IF(PWM_Y39_SET<=300)THEN
	PWM_Y39_SET :=0;
END_IF
IF(PWM_Y40_SET<=300)THEN
	PWM_Y40_SET :=0;
END_IF

END_PROGRAM

// StandardPLC/Application/SaveEngine/SaveEngineMode_12
PROGRAM SaveEngineMode_12
VAR
	PAR_Y1_PosFull:UINT:=600;
END_VAR

(*******************节能控制阀主阀主泵输出执行**************************)
	
//ELSIF(GVL_SaveEngine.SaveEngineMode=12)THEN//节能下降回至中位模式,
	//GVL_SaveEngine.Y72OutPutState:=0;
	//GVL_SaveEngine.Y71OutPutState:=0;
	(****先关Y72再关Y71减少回中位时M1压力冲击****)
GVL_SaveEngine.Y72OutPutState:=0;
IF Mode12Timer>0 THEN
	GVL_SaveEngine.Y71OutPutState:=0;
END_IF
	Y73:=TRUE;
	
PWM_Y7_SET_Target:=0;
PWM_Y9_SET_Target:=0;
PWM_Y8_SET_Target:=0;
PWM_Y10_SET_Target:=0;
RAMP7(
	IN:=WORD_TO_INT(PWM_Y7_SET_Target), 
	ASCEND:= R_RAMP_mainwinch, 
	DESCEND:= F_RAMP_mainwinch_up, 
	TIMEBASE:=TIMEBASE_mainwinch , 
	RESET:=FALSE , 
	OUT=>(PWM_Y7_SET_Target1));
IF(PWM_Y7_SET_Target1>=400) THEN
	Curve_input:=TO_UINT(PWM_Y7_SET_Target1 - 400);
	IF(Curve_input>900) THEN
		Curve_input:=900;
	END_IF
	curve7(input:=REAL_TO_UINT(UINT_TO_REAL(Curve_input)*72.8),Zero:=FALSE,Full:=FALSE,
		   PAR_Progression:=Curve_Par,OutputEnable:=TRUE);
	PWM_Y7_SET:=PAR_Valve1_NegFull + REAL_TO_UINT(UINT_TO_REAL(curve7.Output)/72.8);
ELSE
	PWM_Y7_SET:=0;
END_IF
	
RAMP8(
	IN:=WORD_TO_INT(PWM_Y8_SET_Target), 
	ASCEND:= R_RAMP_mainwinch, 
	DESCEND:= F_RAMP_mainwinch_down, 
	TIMEBASE:=TIMEBASE_mainwinch , 
	RESET:=FALSE , 
	OUT=>(PWM_Y8_SET_Target1));
IF(PWM_Y8_SET_Target1>=400) THEN
	Curve_input:=TO_UINT(PWM_Y8_SET_Target1 - 400);
	IF(Curve_input>900) THEN
		Curve_input:=900;
	END_IF
	curve8(input:=REAL_TO_UINT(UINT_TO_REAL(Curve_input)*72.8),Zero:=FALSE,Full:=FALSE,
		   PAR_Progression:=Curve_Par,OutputEnable:=TRUE);
	PWM_Y8_SET:=PAR_Valve1_NegFull + REAL_TO_UINT(UINT_TO_REAL(curve8.Output)/72.8);
ELSE
	PWM_Y8_SET:=0;
END_IF
	RAMP9(
	IN:=WORD_TO_INT(PWM_Y9_SET_Target), 
	ASCEND:= R_RAMP_mainwinch, 
	DESCEND:= F_RAMP_mainwinch_up, 
	TIMEBASE:=TIMEBASE_mainwinch , 
	RESET:=FALSE , 
	OUT=>(PWM_Y9_SET_Target1));
IF(PWM_Y9_SET_Target1>=400) THEN
	Curve_input:=TO_UINT(PWM_Y9_SET_Target1 - 400);
	IF(Curve_input>900) THEN
		Curve_input:=900;
	END_IF
	curve9(input:=REAL_TO_UINT(UINT_TO_REAL(Curve_input)*72.8),Zero:=FALSE,Full:=FALSE,
		   PAR_Progression:=Curve_Par,OutputEnable:=TRUE);
	PWM_Y9_SET:=PAR_Valve1_NegFull + REAL_TO_UINT(UINT_TO_REAL(curve9.Output)/72.8);
ELSE
	PWM_Y9_SET:=0;
END_IF

RAMP10(
	IN:=WORD_TO_INT(PWM_Y10_SET_Target), 
	ASCEND:= R_RAMP_mainwinch, 
	DESCEND:= F_RAMP_mainwinch_down, 
	TIMEBASE:=TIMEBASE_mainwinch , 
	RESET:=FALSE , 
	OUT=>(PWM_Y10_SET_Target1));
IF(PWM_Y10_SET_Target1>=400) THEN
	Curve_input:=TO_UINT(PWM_Y10_SET_Target1 - 400);
	IF(Curve_input>900) THEN
		Curve_input:=900;
	END_IF
	curve10(input:=REAL_TO_UINT(UINT_TO_REAL(Curve_input)*72.8),Zero:=FALSE,Full:=FALSE,
		   PAR_Progression:=Curve_Par,OutputEnable:=TRUE);
	PWM_Y10_SET:=PAR_Valve1_NegFull + REAL_TO_UINT(UINT_TO_REAL(curve10.Output)/72.8);
ELSE
	PWM_Y10_SET:=0;
END_IF
//Y7 8 9 10范围限制
IF(PWM_Y7_SET>1300)THEN
	PWM_Y7_SET :=1300;
END_IF
IF(PWM_Y8_SET>1300)THEN
	PWM_Y8_SET :=1300;
END_IF
IF(PWM_Y9_SET>1300)THEN
	PWM_Y9_SET :=1300;
END_IF
IF(PWM_Y10_SET>1300)THEN
	PWM_Y10_SET :=1300;
END_IF

IF(PWM_Y7_SET<=300)THEN
	PWM_Y7_SET :=0;
END_IF
IF(PWM_Y8_SET<=300)THEN
	PWM_Y8_SET :=0;
END_IF
IF(PWM_Y9_SET<=300)THEN
	PWM_Y9_SET :=0;
END_IF
IF(PWM_Y10_SET<=300)THEN
	PWM_Y10_SET :=0;
END_IF
	
	
DOH_Y56:=FALSE;
PWM_Y33_SET_Target:=417;//110排量
PWM_Y33_SET := PWM_Y33_SET_Target;
//PWM_Y7_SET:=0;
//PWM_Y9_SET:=0;
//PWM_Y8_SET:=0;
//PWM_Y10_SET:=0;
PWM_Y1_SET:=0;//PWM_Y1_Target 直接给输出 去除中间变量
PWM_Y2_SET:=0; //PWM_Y2_Target 

PWM_Y39_SET_Target:=0;
PWM_Y40_SET_Target:=0;
RAMP19(
IN:=WORD_TO_INT(PWM_Y39_SET_Target), 
ASCEND:= R_RAMP_xiehe, 
DESCEND:= F_RAMP_xiehe, 
TIMEBASE:=TIMEBASE_xiehe , 
RESET:=FALSE , 
OUT=>(PWM_Y39_SET_Target1));
IF(PWM_Y39_SET_Target1>=400) THEN
Curve_input:=TO_UINT(PWM_Y39_SET_Target1 - 400);
IF(Curve_input>900) THEN
	Curve_input:=900;
END_IF
curve19(input:=REAL_TO_UINT(UINT_TO_REAL(Curve_input)*72.8),Zero:=FALSE,Full:=FALSE,
	   PAR_Progression:=Curve_Par1,OutputEnable:=TRUE);
PWM_Y39_SET:=PAR_Valve1_NegFull + REAL_TO_UINT(UINT_TO_REAL(curve19.Output)/72.8);
ELSE
PWM_Y39_SET:=0;
END_IF


RAMP20(
IN:=WORD_TO_INT(PWM_Y40_SET_Target), 
ASCEND:= R_RAMP_xiehe, 
DESCEND:= F_RAMP_xiehe, 
TIMEBASE:=TIMEBASE_xiehe , 
RESET:=FALSE , 
OUT=>(PWM_Y40_SET_Target1));
IF(PWM_Y40_SET_Target1>=400) THEN
Curve_input:=TO_UINT(PWM_Y40_SET_Target1 - 400);
IF(Curve_input>900) THEN
	Curve_input:=900;
END_IF
curve20(input:=REAL_TO_UINT(UINT_TO_REAL(Curve_input)*72.8),Zero:=FALSE,Full:=FALSE,
	   PAR_Progression:=Curve_Par1,OutputEnable:=TRUE);
PWM_Y40_SET:=PAR_Valve1_NegFull + REAL_TO_UINT(UINT_TO_REAL(curve20.Output)/72.8);
ELSE
PWM_Y40_SET:=0;
END_IF

IF(PWM_Y39_SET>1300)THEN
PWM_Y39_SET :=1300;
END_IF
IF(PWM_Y40_SET>1300)THEN
PWM_Y40_SET :=1300;
END_IF

IF(PWM_Y39_SET<=300)THEN
PWM_Y39_SET :=0;
END_IF
IF(PWM_Y40_SET<=300)THEN
PWM_Y40_SET :=0;
END_IF

(*
PWM_Y8_SET:=REAL_TO_UINT(INT_TO_REAL(PWM_JOYY_L_UP_1)/1000*(PAR_Valve1_PosFull-PAR_Valve1_NegFull)+PAR_Valve1_NegFull);
PWM_Y10_SET:=REAL_TO_UINT(INT_TO_REAL(PWM_JOYY_L_UP_1)/1000*(PAR_Valve2_PosFull-PAR_Valve2_NegFull)+PAR_Valve2_NegFull);
PWM_Y1_Target:=REAL_TO_UINT(INT_TO_REAL(PWM_JOYY_L_UP_1)/1000*(PAR_Y1_PosFull-PAR_Y1_NegFull)+PAR_Y1_NegFull);
PWM_Y2_Target:=REAL_TO_UINT(INT_TO_REAL(PWM_JOYY_L_UP_1)/1000*(PAR_Y1_PosFull-PAR_Y2_NegFull)+PAR_Y2_NegFull);
*)
(*  //Y33输出处理
IF PWM_Y33_SET>=PWM_Y33_SET_Target THEN
PWM_Y33_SET := PWM_Y33_SET_Target;
END_IF
	
IF(PWM_Y33_SET<PWM_Y33_SET_Target) THEN
	PWM_Y33_SET:=REAL_TO_UINT(UINT_TO_REAL(PWM_Y33_SET)+JianGE6);
END_IF

IF DIL_SQ3 THEN
	PWM_Y33_SET:=0;
END_IF
*)	
(*主泵功率控制*)

//区分发动机转速
MainPump_Pressure_Taget1450:=PAR_NegFull_x;
MainPump_Pressure_Taget1600:=PAR_PosFull_x;
MainPump_Pressure_Taget1750:=PAR_Zero_x;
IF EngineSpeedTarget<=1080 THEN SPEED_CASE:=1;
ELSIF EngineSpeedTarget>1080 AND EngineSpeedTarget<=1300 THEN SPEED_CASE:=2;
ELSIF EngineSpeedTarget>1300 AND EngineSpeedTarget<=1520 THEN SPEED_CASE:=3;
ELSIF EngineSpeedTarget>1520 AND EngineSpeedTarget<=1680 THEN SPEED_CASE:=4;
ELSIF EngineSpeedTarget>1680 AND EngineSpeedTarget<=1820 THEN SPEED_CASE:=5;
ELSIF EngineSpeedTarget>1820 THEN SPEED_CASE:=6;;END_IF
//不同转速下的发动机最大功率*)
CASE SPEED_CASE OF
1:  Enginer_Power:=135;
2:  Enginer_Power:=174;
3:  Enginer_Power:=200;
4:  Enginer_Power:=230;
5:  Enginer_Power:=250;
6:  Enginer_Power:=261;
END_CASE
//不同转速下的压力值
IF(CANO_Fubeng_Press>100)THEN
	CASE SPEED_CASE OF
	1:MainPump_Pressure_Taget:=MainPump_Pressure_Taget1000-HELIU_Press_Target1000;
	2:MainPump_Pressure_Taget:=MainPump_Pressure_Taget1200-HELIU_Press_Target1200;
	3:MainPump_Pressure_Taget:=MainPump_Pressure_Taget1450-HELIU_Press_Target1400;
	4:MainPump_Pressure_Taget:=MainPump_Pressure_Taget1600-HELIU_Press_Target1600;
	5:MainPump_Pressure_Taget:=MainPump_Pressure_Taget1750-HELIU_Press_Target1800;
	6:MainPump_Pressure_Taget:=MainPump_Pressure_Taget1900-HELIU_Press_Target1900;
	END_CASE
ELSE
	CASE SPEED_CASE OF
	1:MainPump_Pressure_Taget:=MainPump_Pressure_Taget1000;
	2:MainPump_Pressure_Taget:=MainPump_Pressure_Taget1200;
	3:MainPump_Pressure_Taget:=MainPump_Pressure_Taget1450;
	4:MainPump_Pressure_Taget:=MainPump_Pressure_Taget1600;
	5:MainPump_Pressure_Taget:=MainPump_Pressure_Taget1750;
	6:MainPump_Pressure_Taget:=MainPump_Pressure_Taget1900;
	END_CASE		
END_IF

IF( CANI_ECOSwitch) THEN
	CASE SPEED_CASE OF
	1:MainPump_Pressure_Taget:=MainPump_Pressure_Taget1000-ECO_Press_Target1000;
	2:MainPump_Pressure_Taget:=MainPump_Pressure_Taget1200-ECO_Press_Target1200;
	3:MainPump_Pressure_Taget:=MainPump_Pressure_Taget1450-ECO_Press_Target1400;
	4:MainPump_Pressure_Taget:=MainPump_Pressure_Taget1600-ECO_Press_Target1600;
	5:MainPump_Pressure_Taget:=MainPump_Pressure_Taget1750-ECO_Press_Target1800;
	6:MainPump_Pressure_Taget:=MainPump_Pressure_Taget1900-ECO_Press_Target1900;
	END_CASE
END_IF
MainPump_Pressure:=CANO_MainPUMP_Press1+CANO_MainPUMP_Press2;
//消除滤波
MainPump_Pressure_Subtract:= UINT_TO_INT(MainPump_Pressure-MainPump_Pressure_last1);


//大范围波动
IF MainPump_Pressure_Subtract>270 OR MainPump_Pressure_Subtract<-270 THEN
	Subtract:=TRUE;
ELSE
	Subtract:=FALSE;	
END_IF
	TIME_LvBo4(IN:=Subtract,PT:=T#10MS);
	
IF(TIME_LvBo4.Q)  AND (CANO_MainPUMP_Press1>210) THEN 
		MainPump_Pressure_ChangeBool1:=TRUE;
END_IF
	TIME_LvBo1(IN:=MainPump_Pressure_ChangeBool1,PT:=T#2S);
IF(TIME_LvBo1.Q) THEN
	MainPump_Pressure_ChangeBool1 :=FALSE;
END_IF

IF(MainPump_Pressure_ChangeBool1) AND (MainPump_Pressure>MainPump_Pressure_last1) THEN 
	MainPump_Pressure_last1:=MainPump_Pressure;
END_IF

//小范围波动
t_powertime:=TO_TIME(PAR_DeadBand_x);
IF (NOT MainPump_Pressure_ChangeBool1) THEN
	IF(MainPump_Pressure_Subtract>40 OR MainPump_Pressure_Subtract<-40)THEN 
		MainPump_Pressure_ChangeBool:=TRUE;
	ELSE
		MainPump_Pressure_ChangeBool:=FALSE;
	END_IF

	TIME_LvBo2(IN:=MainPump_Pressure_ChangeBool,PT:=t_powertime);
	IF(TIME_LvBo2.Q )THEN
		MainPump_Pressure_last1:=MainPump_Pressure;
	END_IF	
END_IF


IF PowerHead_move AND NOT(MainWinch_move) THEN
		JianGE2:=0.005;
ELSE
	IF(EngineSpeedTarget>1000 AND EngineSpeedTarget<1300)THEN
		JianGE2:=0.005;
	ELSE
		JianGE2:=0.005;
	END_IF
END_IF


IF MainPump_Pressure_last1>MainPump_Pressure_Taget THEN
	Pressure_Coe_Taget:=UINT_TO_REAL(MainPump_Pressure_Taget)/UINT_TO_REAL(MainPump_Pressure_last1);(*压力系数*)
ELSE
	Pressure_Coe_Taget:=1;
END_IF
Pressure_Coe := Pressure_Coe_Taget;


Pressure_Coe := 1;
IF MainPump_Pressure_last1>MainPump_Pressure_Taget  THEN
	IF(PWM_Y1_Target>=PAR_Y1_1_NegFull)THEN
		PWM_Y1_Target_OutPut:=REAL_TO_UINT(UINT_TO_REAL(PWM_Y1_Target-PAR_Y1_1_NegFull)*Pressure_Coe+PAR_Y1_1_NegFull);
	END_IF
	IF(PWM_Y2_Target>=PAR_Y1_1_NegFull)THEN
		PWM_Y2_Target_OutPut:=REAL_TO_UINT(UINT_TO_REAL(PWM_Y2_Target-PAR_Y1_1_NegFull)*Pressure_Coe+PAR_Y1_1_NegFull);
	END_IF
ELSE
	PWM_Y1_Target_OutPut:=PWM_Y1_Target;
	PWM_Y2_Target_OutPut:=PWM_Y2_Target;
END_IF

//PWM_Y1_Target_OutPut:=PWM_Y1_Target;
//PWM_Y2_Target_OutPut:=PWM_Y2_Target;
IF(EngineSpeedTarget>CANO_SPEED AND CANO_SPEED>400)THEN
	EngineSpeedSub:=EngineSpeedTarget - CANO_SPEED;
ELSE
	EngineSpeedSub:=0;
END_IF

IF(PWM_Y1_Target_OutPut<300)THEN PWM_Y1_Target_OutPut:=300;END_IF	
IF(PWM_Y2_Target_OutPut<300)THEN PWM_Y2_Target_OutPut:=300;END_IF

RAMP15_IN:=PWM_Y1_Target_OutPut;
RAMP16_IN:=PWM_Y2_Target_OutPut;
(*
IF MainWinch_move  OR  LeftMove_move OR RightMove_move THEN  
	TIMEBASE_pump:=T#1000MS;
	TIMEBASE_xiehe:=T#500MS;
ELSE
	TIMEBASE_pump:=T#400MS;
	TIMEBASE_xiehe:=T#200MS;
END_IF
t_PowerHead_move(IN:= MainWinch_move,PT:=T#2S);
IF t_PowerHead_move.Q THEN
	F_RAMP_pump:=x_t_PowerHead_move;
	R_RAMP_pump:=x2_t_PowerHead_move;
ELSE
	F_RAMP_pump:=1000;
	R_RAMP_pump:=300;
END_IF
*)
(*  12模式不需要斜坡
RAMP15(
	IN:=UINT_TO_INT(RAMP15_IN), 
	ASCEND:= 300, 
	DESCEND:= 300, 
	TIMEBASE:=T#1000MS , 
	RESET:=FALSE , 
	OUT=>(PWM_Y1_SET));
	
RAMP16(
	IN:=UINT_TO_INT(RAMP16_IN), 
	ASCEND:= 300, 
	DESCEND:= 300, 
	TIMEBASE:=T#1000MS , 
	RESET:=FALSE , 
	OUT=>(PWM_Y2_SET));

*)

	CASE SPEED_CASE OF
                1:F_RAMP_pump:=1500; R_RAMP_pump:=100;                  
                2: 		IF MainWinch_move AND (JiaYa_move OR CANO_JiayaPressure>80)  THEN    //3泵同时起压时，降低主泵的加载速度，避免掉速熄火
                                F_RAMP_pump:=1500; R_RAMP_pump:=100;
                        ELSE
                                F_RAMP_pump:=1500; R_RAMP_pump:=100;//从200降
                                IF  PWM_JOYY_L_UP>10 THEN
                                 F_RAMP_pump:=1500; R_RAMP_pump:=200;
                                END_IF
                        END_IF            
                3:
                        IF MainWinch_move AND (JiaYa_move OR CANO_JiayaPressure>80)  THEN    //3泵同时起压时，降低主泵的加载速度，避免掉速熄火
                                F_RAMP_pump:=1500; R_RAMP_pump:=150;
                        ELSE
                                F_RAMP_pump:=1500; R_RAMP_pump:=TO_INT(PAR_NegFull_y);
                                IF  PWM_JOYY_L_UP>10 THEN
                                 F_RAMP_pump:=1500; R_RAMP_pump:=300;
                                END_IF
                        END_IF                
                4:
                        IF MainWinch_move AND (JiaYa_move OR CANO_JiayaPressure>80)  THEN
                                F_RAMP_pump:=1500; R_RAMP_pump:=150;
                        ELSE
                                F_RAMP_pump:=1500; R_RAMP_pump:=TO_INT(PAR_PosFull_y);//从200降
                                IF  PWM_JOYY_L_UP>10 THEN
                                 F_RAMP_pump:=1500; R_RAMP_pump:=300;
                                END_IF
                        END_IF                                
                5:
                        IF MainWinch_move AND (JiaYa_move OR CANO_JiayaPressure>80)  THEN
                                F_RAMP_pump:=1500; R_RAMP_pump:=200;
                        ELSE
                                F_RAMP_pump:=1500; R_RAMP_pump:=TO_INT(PAR_Zero_y);
                                IF  PWM_JOYY_L_UP>10 THEN
                                 F_RAMP_pump:=1500; R_RAMP_pump:=300;
                                END_IF
                        END_IF                        
                6:		IF MainWinch_move AND (JiaYa_move OR CANO_JiayaPressure>80)  THEN
                                F_RAMP_pump:=1500; R_RAMP_pump:=200;
                        ELSE
                                F_RAMP_pump:=1500; R_RAMP_pump:=200;
                                IF  PWM_JOYY_L_UP>10 THEN
                                 F_RAMP_pump:=1500; R_RAMP_pump:=300;
                                END_IF
                        END_IF	
	END_CASE
(******斜坡增步长300 斜坡降步长300->400*****)	
RAMP15(
	IN:=UINT_TO_INT(RAMP15_IN), 
	ASCEND:= R_RAMP_pump, 
	DESCEND:= 1500, 
	TIMEBASE:=T#1000MS , 
	RESET:=FALSE , 
	OUT=>(PWM_Y1_SET));
(******减斜坡300->400*****)	
RAMP16(
	IN:=UINT_TO_INT(RAMP16_IN), 
	ASCEND:= R_RAMP_pump, 
	DESCEND:= 1500, 
	TIMEBASE:=T#1000MS , 
	RESET:=FALSE , 
	OUT=>(PWM_Y2_SET));

IF (NOT Rotation_move) AND (NOT MainWinch_move) AND (NOT PowerHead_move)
		AND (NOT JiaYa_move) AND (NOT ViceWinch_move)
		AND (NOT LeftMove_move) AND (NOT RightMove_move)  THEN
	PWM_Y1_Target:=0;
	PWM_Y2_Target:=0;
END_IF

IF PWM_Y1_SET<TO_INT(PAR_Y1_1_NegFull )THEN
	PWM_Y1_SET:=TO_INT(PAR_Y1_1_NegFull);
END_IF

IF PWM_Y2_SET<TO_INT(PAR_Y1_1_NegFull )THEN
	PWM_Y2_SET:=TO_INT(PAR_Y1_1_NegFull);
END_IF

IF(PWM_Y1_SET>1000) THEN
	PWM_Y1_SET := 300;
END_IF

IF(PWM_Y2_SET>1000) THEN
	PWM_Y2_SET := 300;
END_IF

END_PROGRAM

// StandardPLC/Application/SaveEngine/SaveEngineMode_9
PROGRAM SaveEngineMode_9
VAR
DI_PWM_JOYX_L: BOOL;
	DI_PWM_JOYY_L: BOOL;
	DI_PWM_JOYX_R: BOOL;
	DI_PWM_JOYY_R: BOOL;
	DI_PWM_JOY_Jiao_R: BOOL;
	DI_PWM_JOY_Jiao_L: BOOL;
	Rotation_move: BOOL;
	MainWinch_move:BOOL;
	PowerHead_move:BOOL;
	JiaYa_move: BOOL;
	LvZhang_move: BOOL;
	BianFu_move:BOOL;
	ViceWinch_move: BOOL;
	LeftMove_move:BOOL;
	RightMove_move:BOOL;
	SPEED_CASE:USINT;
	Enginer_Power:UINT;
	
	PWM_Y1_Target: UINT;	
	PWM_Y2_Target: UINT;	
	
	PWM_Y1_Target_MAX: UINT;
	PWM_Y2_Target_MAX: UINT;
	Hydraulic_Power2:UINT;
	Hydraulic_Power1:UINT;
	Hydraulic_Power:UINT;
	Enginer_Rat: UINT;
	MainPump_Pressure_Taget:UINT;
	Coe_valve: REAL;	
	MainPump_Pressure: UINT;
	Pressure_Coe: REAL;
	PWM_Y1_Target_1: UINT;
	Single_move:BOOL;
	PWM_Y1_Target_OutPut: UINT;
	PWM_Y2_Target_OutPut: UINT;
	PWM_Y34_SET_Target: UINT:=0;
	PWM_Y33_SET_Target: UINT:=1100;
	

	DonglitouBlink:BLINK;
	DonglitouBlink_biaozhi:BOOL;
	DOH_Y50_1: BOOL;
	Rotation_late:TOF;
	MainPump_Pressure_Taget1000:UINT:=220;
	MainPump_Pressure_Taget1200:UINT:=360;
	MainPump_Pressure_Taget1450:UINT:=420;
	MainPump_Pressure_Taget1600:UINT:=420;
	MainPump_Pressure_Taget1750:UINT:=400;
	MainPump_Pressure_Taget1900:UINT:=360;
	Pressure_Coe_Taget: REAL;
	JianGE1: REAL:=1;
	JianGE2: REAL:=0.005;
	JianGE3: REAL:=3;
	TIME_100ms:TON;
	MainPump_Pressure_last: UINT;
	MainPump_Pressure_last1: UINT;
	TIME_LvBo1:TON;
	TIME_LvBo2:TON;
	TIME_LvBo3:TON;
	MainPump_Pressure_Subtract: INT;
	MainPump_Pressure_ChangeBool: BOOL;
	MainPump_Pressure_ChangeBool1:BOOL;
	PWM_Y2_Target_fuhe: UINT;
	PWM_Y1_Target_fuhe: UINT;
	EngineSpeedSub: UINT;
	PWM_Y23_SET_Taget: UINT;
	PWM_Y24_SET_Taget: UINT;
	CANO_DonglitouPressure_last: UINT;
	DonglitouPressureSub:INT;
	DonglitouPressure_ChangeBool: BOOL;
	JieSuoBool: BOOL;
	ECO_Press_Target1000: UINT:=50;
	ECO_Press_Target1200: UINT:=50;
	ECO_Press_Target1400: UINT:=50;
	ECO_Press_Target1600: UINT:=50;
	ECO_Press_Target1800: UINT:=50;
	ECO_Press_Target1900: UINT:=50;
	
	HELIU_Press_Target1000: UINT:=80;
	HELIU_Press_Target1200: UINT:=80;
	HELIU_Press_Target1400: UINT:=80;
	HELIU_Press_Target1600: UINT:=80;
	HELIU_Press_Target1800: UINT:=80;
	HELIU_Press_Target1900: UINT:=80;
	PWM_Y2_Target_P: UINT;
	PWM_JOY_P_W: UINT;
	XISHU1: REAL:=0.6;
	BiaoZHI_MainWinchUp: BOOL;
	JianGE6:REAL:=2;
	PWM_Y5_SET_Target: UINT;
	PWM_Y6_SET_Target: UINT;
	PWM_Y15_SET_Target: UINT;
	PWM_Y16_SET_Target: UINT;
	PWM_Y5_SET_Target1: INT;
	PWM_Y6_SET_Target1: INT;
	PWM_Y15_SET_Target1: INT;
	PWM_Y16_SET_Target1: INT;
	PWM_Y8_SET_Target: UINT;
	PWM_Y10_SET_Target: UINT;
	PWM_Y7_SET_Target: UINT;
	PWM_Y9_SET_Target: UINT;
	PWM_Y8_SET_Target1: INT;
	PWM_Y10_SET_Target1: INT;
	PWM_Y7_SET_Target1: INT;
	PWM_Y9_SET_Target1: INT;
	JianGE7: UINT:=20;
	JianGE8: UINT:=3;
	PWM_Y39_SET_Target: UINT;
	PWM_Y40_SET_Target: UINT;
	ABS_JOY_1: INT;
	PWM_Y61_SET_Tatget: UINT;
	PWM_Y12_SET_Tatget: UINT;
	PWM_Y14_SET_Tatget: UINT;
	PWM_Y60_SET_Tatget: UINT;
	PWM_Y11_SET_Tatget: UINT;
	PWM_Y13_SET_Tatget: UINT;
	PWM_Y61_SET_Tatget1: INT;
	PWM_Y12_SET_Tatget1: INT;
	PWM_Y14_SET_Tatget1: INT;
	PWM_Y60_SET_Tatget1: INT;
	PWM_Y11_SET_Tatget1: INT;
	PWM_Y13_SET_Tatget1: INT;
	JianGE10: UINT:=25;
	yyyy: UINT;
	TIME_200ms:TON;
	TIME_400ms:TON;
	CANI_JOYX_R_last:UINT;
	Sub_Joyx_r: INT;
	Joyx_change_bool: BOOL;
	JianGE12: UINT:=30;
	Sub_Joyx_r_1: INT;
	BIAOzhi1: BOOL;
	R_TRIG_1:R_TRIG;
	R_TRIG_BOOL: BOOL;
	JianGE22: REAL;
	
	
	curve:curve_quxian;
	curve1:curve_quxian;
	curve2:curve_quxian;
	curve3:curve_quxian;
	curve4:curve_quxian;
	curve5:curve_quxian;
	curve6:curve_quxian;
	curve7:curve_quxian;
	curve8:curve_quxian;
	curve9:curve_quxian;
	curve10:curve_quxian;
	curve11:curve_quxian;
	curve12:curve_quxian;
	curve13:curve_quxian;
	curve14:curve_quxian;
	curve19:curve_quxian;
	curve20:curve_quxian;
	COUNTER : INT;
	JianGE13: UINT:=40;
	JianGE14: UINT:=40;
	RAMP:RAMP_INT;
	RAMP1:RAMP_INT;
	RAMP2:RAMP_INT;
	RAMP3:RAMP_INT;
	R_RAMP:INT:=400;
	F_RAMP:INT:=250;
	TIMEBASE:TIME:=T#200MS;
	PWM_Y7_SET_Target111: INT;
	YYYYYYY:BOOL;
	JIANGE1111: INT:=20;
	
	RAMP4:RAMP_INT;
	RAMP5:RAMP_INT;
	RAMP6:RAMP_INT;
	RAMP7:RAMP_INT;
	RAMP8:RAMP_INT;
	RAMP9:RAMP_INT;
	RAMP10:RAMP_INT;
	RAMP11:RAMP_INT;
	RAMP12:RAMP_INT;
	RAMP13:RAMP_INT;
	RAMP14:RAMP_INT;
	RAMP15:RAMP_INT;
	RAMP16:RAMP_INT;
	RAMP17:RAMP_INT;
	RAMP18:RAMP_INT;
	RAMP19:RAMP_INT;
	RAMP20:RAMP_INT;
	RAMP21:RAMP_INT;
	RAMP22:RAMP_INT;
	RAMP23:RAMP_INT;
	RAMP24:RAMP_INT;
	PWM_Y23_SET_Taget1:INT;
	PWM_Y24_SET_Taget1:INT;
	PWM_Y18_SET_Taget1:INT;
	PWM_Y18_SET_Taget:UINT;
	ASCEND_value2:INT;
	//2023 01 13 增加
	//行走动作斜坡值
	R_RAMP_traval:INT:=800;
	F_RAMP_traval:INT:=400;
	TIMEBASE_traval:TIME:=T#200MS;
	//动力头动作斜坡值
	R_RAMP_ratate:INT:=800;
	F_RAMP_ratate:INT:=800;
	TIMEBASE_ratate:TIME:=T#100MS;
	//主卷扬动作斜坡值
	R_RAMP_mainwinch:INT:=800;
	F_RAMP_mainwinch_up:INT:=400;
	F_RAMP_mainwinch_down:INT:=400;
	TIMEBASE_mainwinch:TIME:=T#200MS;
	//主泵排量斜坡值
	R_RAMP_pump:INT:=300;
	F_RAMP_pump:INT:=1000;
	TIMEBASE_pump:TIME:=T#1000MS;
	//卸荷阀斜坡值
	R_RAMP_xiehe:INT:=500;
	F_RAMP_xiehe:INT:=400;
	TIMEBASE_xiehe:TIME:=T#500MS;
	
	//直线阀斜坡值
	R_RAMP_zhixian:INT:=800;
	F_RAMP_zhixian:INT:=800;
	TIMEBASE_zhixian:TIME:=T#300MS;
		
	Subtract: BOOL;
	TIME_LvBo4:TON;
	Curve_input:UINT;
	Curve_Par: SINT:=0;
	Curve_Par1: SINT:=0;
	Move_JOY_FUHE: UINT;
	PWM_JOY_Jiao_L_UP1:UINT;
	PWM_JOY_Jiao_L_DOWN1:UINT;
	PWM_JOY_Jiao_R_UP1:UINT;
	PWM_JOY_Jiao_R_DOWN1:UINT;
	
	PWM_JOYX_R_UP_a:UINT;
	PWM_JOYX_R_UP_b:UINT;
	
	PWM_JOYX_R_DOWN_a:UINT;
	PWM_JOYX_R_DOWN_b:UINT;
	
	PWM_JOYY_L_DOWN_a:UINT;
	PWM_JOYY_L_DOWN_b:UINT;
	
	PWM_JOYY_L_UP_a:UINT;
	PWM_JOYY_L_UP_b:UINT;
	aaaa:UINT:=500;
	
	JOY_PAOTU:BOOL;
	
	JOY_PAOTU_tiaojian:BOOL;
	TIME_1000_1ms:ton;
	tempbool:BOOL;
	CANI_JOYX_R_last2:UINT;
	Sub_Joyx_r2:INT;
	JianGE11:REAL:=2;
	JianGE21:uint:=10;
	END_IFc: INT;
	x1:UINT:=8;
	x2:UINT:=8;
	PWM_JOY_JIAO:UINT;
	PWM_Y39_SET1:UINT;
	PWM_Y40_SET1:UINT;
	aaa: INT;
	TIME_50ms:TON;
	TIME_55ms:TOF;
	TIME_2000ms:TOF;
	start_move: BOOL;
	T1:TIME;
	TEMP1:UINT;
	X3: INT;
	X4: INT;
	liandong:BOOL;
	PWM_Y9_SET1:INT;
	PWM_Y10_SET1:INT;
	PWM_Y13_SET1:INT;
	PWM_Y14_SET1:INT;
	yanchi1:BOOL;
	yanchi_ton1:ton;
	RAMP15_IN:UINT;
	RAMP16_IN:UINT;
	Rtrig_d1:R_TRIG;
	Rtrig_d2:R_TRIG;
	
	Rtrig_DongLiTou1:R_TRIG;
	Rtrig_DongLiTou2:R_TRIG;
	Count_TIMES_Fanzhuan: UINT;
	Count_TIMES_Zhengzhuan: UINT;
	TIME_1000ms:TON;
	TIME_1000ms_TP:TON;
	Count_TIMES_Fanzhuan_LAST: UINT;
	Count_TIMES_Zhengzhuan_LAST: UINT;
	Paotu_Modle: BOOL;
	PaoTU_biaozhi: BOOL;
	TIMEBASE_D: TIME;
	PWM_Y39_SET_Target1:INT;
	PWM_Y40_SET_Target1:INT;
	PWM_Y37_SET_Target:UINT;
	PWM_Y17_SET2:UINT;
	t_PowerHead_move:TON;
	x_t_PowerHead_move:INT:=10;//100-10
	x2_t_PowerHead_move:INT:=10;//100-10
	P_value:REAL;//动力头反转+主卷上提时的分流系数
	PWM_JOY_P:UINT;
	PWM_JOY_P1:UINT;
	PWM_JOY_P2:UINT;
	PWM_JOY_P3:UINT;
	PWM_JOY_P4:UINT;
	ASCEND_value:INT;
	ftp1:INT:=500;
	ftp2:INT:=100;
	t_powertime:TIME;
	
	P25_Flag:BOOL;
	P27_Flag:BOOL;
	P29_Flag:BOOL;
	P31_Flag:BOOL;
	PressLvBo_TON:TON;
	PressLvBo_TON1: TON;
	PressLvBo_TON2: TON;
	PressLvBo_TON3: TON;
	test: BYTE;
	testpaotu: UINT := 450;
END_VAR

//动力头反转与主卷上提时的分流系数值
(*IF CANO_ZhuJuanPressure<=100 THEN
	P_value:=TO_REAL(PAR_KI+40)/100.0;
ELSIF CANO_ZhuJuanPressure>100 AND  CANO_ZhuJuanPressure<=200 THEN
	P_value:=TO_REAL(PAR_KI+20)/100.0;
ELSE
	P_value:=TO_REAL(PAR_KI)/100;
END_IF*)
GVL_SaveEngine.Y72OutPutState:=0;
GVL_SaveEngine.Y71OutPutState:=0;
GVL_SaveEngine.Y73:=0;
P_value:=TO_REAL(PAR_KI)/100;  //出厂值设定为35
//喇叭
IF DI_LHandle_SB5 THEN
	DOH_Y59:=TRUE;
ELSE
	DOH_Y59:=FALSE;
END_IF
//延时断电
TIME_2000ms(IN:=DIH_power3,PT:=T#2S);
IF(TIME_2000ms.Q)THEN
	DOH_YS3:=TRUE;
ELSE
	DOH_YS3:=FALSE;
END_IF

//主卷上限位及解锁
IF(DI_LHandle_SB1 AND (NOT CANI_WorkModeSwitch))THEN
	JieSuoBool:=TRUE;
ELSE
	JieSuoBool:=FALSE;	
END_IF

IF DIL_SQ4 THEN
	IF(NOT JieSuoBool) THEN
		PWM_JOYY_L_DOWN:=0;
	END_IF
END_IF

//主卷下限位及解锁
//主卷下放限制
IF( CANO_MainWinchTension*100<PAR_MainWinchLaLi_Low) AND (NOT DI_LHandle_SB1) AND (CANI_WorkModeSwitch)THEN
	PWM_JOYY_L_UP:=0;
END_IF

TIME_50ms(in:=start_move,pt:=T1);
TIME_55ms(in:=start_move,pt:=T#500MS);
IF( LeftMove_move OR  RightMove_move  OR   MainWinch_move OR PowerHead_move OR ViceWinch_move )THEN
	start_move:=TRUE;
ELSE
	start_move:=FALSE;
END_IF
	 


IF NOT DIL_SQ3 THEN(*先导控制输入*)
	IF PWM_JOYX_L_UP>10 OR PWM_JOYX_L_DOWN>10 THEN  DI_PWM_JOYX_L := TRUE;ELSE DI_PWM_JOYX_L:=FALSE;END_IF(*左手柄左右动作*)
	IF PWM_JOYY_L_UP>10 OR PWM_JOYY_L_DOWN>10 THEN  DI_PWM_JOYY_L := TRUE;ELSE DI_PWM_JOYY_L:=FALSE;END_IF(*左手柄前后动作*)
	IF PWM_JOYX_R_UP>10 OR PWM_JOYX_R_DOWN>10 THEN  DI_PWM_JOYX_R := TRUE;ELSE DI_PWM_JOYX_R:=FALSE;END_IF(*右手柄左右动作*)
	IF PWM_JOYY_R_UP>10 OR PWM_JOYY_R_DOWN>10 THEN  DI_PWM_JOYY_R := TRUE;ELSE DI_PWM_JOYY_R:=FALSE;END_IF(*右手柄前后动作*)
	IF PWM_JOY_Jiao_L_UP>10 OR PWM_JOY_Jiao_L_DOWN>10 THEN  DI_PWM_JOY_Jiao_L:= TRUE;ELSE DI_PWM_JOY_Jiao_L:=FALSE;END_IF(*左脚踏前后动作*)
	IF PWM_JOY_Jiao_R_UP>10 OR PWM_JOY_Jiao_R_DOWN>10 THEN  DI_PWM_JOY_Jiao_R := TRUE;ELSE DI_PWM_JOY_Jiao_R:=FALSE;END_IF(*左脚踏左右动作*)
ELSE
	DI_PWM_JOYX_L:=FALSE;
	DI_PWM_JOYY_L:=FALSE;
	DI_PWM_JOYX_R:=FALSE;
	DI_PWM_JOYY_R:=FALSE;
	DI_PWM_JOY_Jiao_L:=FALSE;
	DI_PWM_JOY_Jiao_R:=FALSE;
END_IF

(*动作标志*)
IF DI_PWM_JOYY_L THEN MainWinch_move:=TRUE; ELSE MainWinch_move:=FALSE;END_IF(*主卷扬动作*)
IF DI_PWM_JOYX_L THEN Rotation_move:=TRUE; ELSE Rotation_move:=FALSE;END_IF(*回转动作*)
IF CANI_WorkModeSwitch THEN   (*作业挡情况下*)
	IF DI_PWM_JOYX_R THEN PowerHead_move:=TRUE;ELSE PowerHead_move:=FALSE;END_IF(*动力头回转动作*)
	IF DI_PWM_JOYY_R THEN JiaYa_move:=TRUE;ELSE JiaYa_move:=FALSE;END_IF(*动力头加压动作*)
	LvZhang_move:=FALSE;
	BianFu_move:=FALSE;
	ViceWinch_move:=FALSE;
	LeftMove_move:=FALSE;
	RightMove_move:=FALSE;
ELSE   (*调整档状态*)
	IF DI_PWM_JOYX_R THEN  LvZhang_move:=TRUE;ELSE LvZhang_move:=FALSE;END_IF(*L履带、张紧、支腿动作,M4阀*)
	(*LeftMove_move:=DI_PWM_JOY_Jiao_L;(*左行走动作*)
	RightMove_move:=DI_PWM_JOY_Jiao_R;*)(*右行走动作*)
	IF( PWM_JOY_Jiao_L_UP1>10 OR PWM_JOY_Jiao_L_DOWN1>10)  AND  DI_PWM_JOY_Jiao_L THEN
		LeftMove_move:=TRUE;
	ELSE
		LeftMove_move:=FALSE;
	END_IF
	IF( PWM_JOY_Jiao_R_UP1>10 OR PWM_JOY_Jiao_R_DOWN1>10)  AND  DI_PWM_JOY_Jiao_R THEN
		RightMove_move:=TRUE;
	ELSE
		RightMove_move:=FALSE;
	END_IF

	IF  DI_RHandle_SB5 THEN
		ViceWinch_move:=FALSE;
		IF  DI_PWM_JOYY_R  THEN BianFu_move:=TRUE;ELSE BianFu_move:=FALSE;END_IF(*变幅动作M4阀*)
	ELSE
		BianFu_move:=FALSE;
		IF DI_PWM_JOYY_R  THEN ViceWinch_move:=TRUE;ELSE ViceWinch_move:=FALSE;END_IF(*副卷扬动作M4阀*)
	END_IF
	PowerHead_move:=FALSE;
	JiaYa_move:=FALSE;
END_IF


(****主阀单动作标志****)
	IF (NOT MainWinch_move) AND (NOT PowerHead_move) AND (ViceWinch_move) THEN
		Single_move:=TRUE;
	ELSE
		Single_move:=FALSE;
	END_IF
	
//先导控制
IF(NOT DIL_SQ3) AND NOT VarGpsSystemLockedState THEN
	DOH_Y51:=TRUE;
ELSE
	DOH_Y51:=FALSE;
END_IF

//行走动作
(*脚踏阀偏差*)
IF   ((PWM_JOY_Jiao_L_UP-PWM_JOY_Jiao_R_UP)<200 OR(PWM_JOY_Jiao_R_UP-PWM_JOY_Jiao_L_UP)<200) THEN
	PWM_JOY_Jiao_L_UP1:=MAX(PWM_JOY_Jiao_L_UP,PWM_JOY_Jiao_R_UP);
	PWM_JOY_Jiao_R_UP1:=MAX(PWM_JOY_Jiao_L_UP,PWM_JOY_Jiao_R_UP);
ELSE
	PWM_JOY_Jiao_L_UP1:=PWM_JOY_Jiao_L_UP;
	PWM_JOY_Jiao_R_UP1:=PWM_JOY_Jiao_R_UP;
END_IF
IF   ((PWM_JOY_Jiao_L_DOWN-PWM_JOY_Jiao_R_DOWN)<200  OR  (PWM_JOY_Jiao_R_DOWN-PWM_JOY_Jiao_L_DOWN)<200 ) THEN
	PWM_JOY_Jiao_L_DOWN1:=MAX(PWM_JOY_Jiao_L_DOWN,PWM_JOY_Jiao_R_DOWN);
	PWM_JOY_Jiao_R_DOWN1:=MAX(PWM_JOY_Jiao_L_DOWN,PWM_JOY_Jiao_R_DOWN);
ELSE
	PWM_JOY_Jiao_L_DOWN1:=PWM_JOY_Jiao_L_DOWN;
	PWM_JOY_Jiao_R_DOWN1:=PWM_JOY_Jiao_R_DOWN;
END_IF

PWM_JOY_JIAO:=MAX(PWM_JOY_Jiao_L_UP1,PWM_JOY_Jiao_R_UP1,PWM_JOY_Jiao_L_DOWN1,PWM_JOY_Jiao_R_DOWN1);
liandong:=FALSE;
(*左行走*)
(*泵1   Y1   Y39控制右行走   Y15  16 *)
(*泵2   Y2 Y40 控制左行走    Y5  Y6*)
IF LeftMove_move THEN
	IF PWM_JOY_Jiao_L_UP1>10 THEN
		PWM_Y2_Target:=REAL_TO_UINT(UINT_TO_REAL(PWM_JOY_Jiao_L_UP1)/1000*(PAR_Y1_1_PosFull-PAR_Y1_1_NegFull)+PAR_Y1_1_NegFull);
		PWM_Y5_SET_Target:=REAL_TO_UINT(UINT_TO_REAL(PWM_JOY_Jiao_L_UP1)/1000*(PAR_Valve2_PosFull-PAR_Valve2_NegFull)+PAR_Valve2_NegFull);
		PWM_Y6_SET_Target:=0;	
	ELSIF PWM_JOY_Jiao_L_DOWN1>10 THEN
		PWM_Y2_Target:=REAL_TO_UINT(UINT_TO_REAL(PWM_JOY_Jiao_L_DOWN1)/1000*(PAR_Y1_1_PosFull-PAR_Y1_1_NegFull)+PAR_Y1_1_NegFull);
		PWM_Y6_SET_Target:=REAL_TO_UINT(UINT_TO_REAL(PWM_JOY_Jiao_L_DOWN1)/1000*(PAR_Valve2_PosFull-PAR_Valve2_NegFull)+PAR_Valve2_NegFull);
		PWM_Y5_SET_Target:=0;		
	END_IF
ELSE
	PWM_Y5_SET_Target:=0;
	PWM_Y6_SET_Target:=0;
END_IF
(*右行走*)
IF RightMove_move  THEN
	IF PWM_JOY_Jiao_R_UP1>10 THEN
		PWM_Y1_Target:=REAL_TO_UINT(UINT_TO_REAL(PWM_JOY_Jiao_R_UP1)/1000*(PAR_Y1_1_PosFull-PAR_Y1_1_NegFull)+PAR_Y1_1_NegFull);
		PWM_Y15_SET_Target:=REAL_TO_UINT(UINT_TO_REAL(PWM_JOY_Jiao_R_UP1)/1000*(PAR_Valve1_PosFull-PAR_Valve1_NegFull)+PAR_Valve1_NegFull);
		PWM_Y16_SET_Target:=0;
	
	ELSIF PWM_JOY_Jiao_R_DOWN1>10 THEN
		PWM_Y1_Target:=REAL_TO_UINT(UINT_TO_REAL(PWM_JOY_Jiao_R_DOWN1)/1000*(PAR_Y1_1_PosFull-PAR_Y1_1_NegFull)+PAR_Y1_1_NegFull);
		PWM_Y16_SET_Target:=REAL_TO_UINT(UINT_TO_REAL(PWM_JOY_Jiao_R_DOWN1)/1000*(PAR_Valve1_PosFull-PAR_Valve1_NegFull)+PAR_Valve1_NegFull);
		PWM_Y15_SET_Target:=0;
		
	END_IF
ELSE
	PWM_Y15_SET_Target:=0;
	PWM_Y16_SET_Target:=0;
END_IF

	//如有必要，可根据行走阀开关大小调整斜坡值
(*	IF(PWM_Y5_SET<1000  AND  PWM_Y5_SET>=900)THEN
			R_RAMP_traval:=100;
	ELSIF(PWM_Y5_SET<900 AND PWM_Y5_SET>=780)THEN
			R_RAMP_traval:=10;
	ELSE
			R_RAMP_traval:=250;
	END_IF
		
	IF(PWM_Y6_SET<1000  AND  PWM_Y6_SET>=900)THEN
			F_RAMP_traval:=100;		
	ELSIF(PWM_Y6_SET<900 AND PWM_Y6_SET>750 )THEN
			F_RAMP_traval:=15;
	ELSE
			F_RAMP_traval:=250;
	END_IF*)
	
(*行走动作缓冲*)
RAMP11(
	IN:=WORD_TO_INT(PWM_Y5_SET_Target), 
	ASCEND:= R_RAMP_traval, 
	DESCEND:= F_RAMP_traval, 
	TIMEBASE:=TIMEBASE_traval , 
	RESET:=FALSE , 
	OUT=>(PWM_Y5_SET_Target1));
IF(PWM_Y5_SET_Target1>=400) THEN
	Curve_input:=TO_UINT(PWM_Y5_SET_Target1 - 400);
	IF(Curve_input>900) THEN
		Curve_input:=900;
	END_IF
	curve11(input:=REAL_TO_UINT(UINT_TO_REAL(Curve_input)*72.8),Zero:=FALSE,Full:=FALSE,
		   PAR_Progression:=Curve_Par1,OutputEnable:=TRUE);
	PWM_Y5_SET:=PAR_Valve1_NegFull + REAL_TO_UINT(UINT_TO_REAL(curve11.Output)/72.8);
ELSE
	PWM_Y5_SET:=0;
END_IF

RAMP12(
	IN:=WORD_TO_INT(PWM_Y6_SET_Target), 
	ASCEND:= R_RAMP_traval, 
	DESCEND:= F_RAMP_traval, 
	TIMEBASE:=TIMEBASE_traval , 
	RESET:=FALSE , 
	OUT=>(PWM_Y6_SET_Target1));
IF(PWM_Y6_SET_Target1>=400) THEN
	Curve_input:=TO_UINT(PWM_Y6_SET_Target1 - 400);
	IF(Curve_input>900) THEN
		Curve_input:=900;
	END_IF
	curve12(input:=REAL_TO_UINT(UINT_TO_REAL(Curve_input)*72.8),Zero:=FALSE,Full:=FALSE,
		   PAR_Progression:=Curve_Par1,OutputEnable:=TRUE);
	PWM_Y6_SET:=PAR_Valve1_NegFull + REAL_TO_UINT(UINT_TO_REAL(curve12.Output)/72.8);
ELSE
	PWM_Y6_SET:=0;
END_IF

RAMP13(
	IN:=WORD_TO_INT(PWM_Y15_SET_Target), 
	ASCEND:= R_RAMP_traval, 
	DESCEND:= F_RAMP_traval, 
	TIMEBASE:=TIMEBASE_traval , 
	RESET:=FALSE , 
	OUT=>(PWM_Y15_SET_Target1));
IF(PWM_Y15_SET_Target1>=400) THEN
	Curve_input:=TO_UINT(PWM_Y15_SET_Target1 - 400);
	IF(Curve_input>900) THEN
		Curve_input:=900;
	END_IF
	curve13(input:=REAL_TO_UINT(UINT_TO_REAL(Curve_input)*72.8),Zero:=FALSE,Full:=FALSE,
		   PAR_Progression:=Curve_Par1,OutputEnable:=TRUE);
	PWM_Y15_SET:=PAR_Valve1_NegFull + REAL_TO_UINT(UINT_TO_REAL(curve13.Output)/72.8);
ELSE
	PWM_Y15_SET:=0;
END_IF

RAMP14(
	IN:=WORD_TO_INT(PWM_Y16_SET_Target), 
	ASCEND:= R_RAMP_traval, 
	DESCEND:= F_RAMP_traval, 
	TIMEBASE:=TIMEBASE_traval , 
	RESET:=FALSE , 
	OUT=>(PWM_Y16_SET_Target1));
IF(PWM_Y16_SET_Target1>=400) THEN
	Curve_input:=TO_UINT(PWM_Y16_SET_Target1 - 400);
	IF(Curve_input>900) THEN
		Curve_input:=900;
	END_IF
	curve14(input:=REAL_TO_UINT(UINT_TO_REAL(Curve_input)*72.8),Zero:=FALSE,Full:=FALSE,
		   PAR_Progression:=Curve_Par1,OutputEnable:=TRUE);
	PWM_Y16_SET:=PAR_Valve1_NegFull + REAL_TO_UINT(UINT_TO_REAL(curve14.Output)/72.8);
ELSE
	PWM_Y16_SET:=0;
END_IF


(*直线行走*)
(*IF(  DIH_SA19)THEN
	IF (PWM_JOY_Jiao_L_UP1>10  AND PWM_JOY_Jiao_R_UP1>10) OR ( PWM_JOY_Jiao_L_DOWN1>10 AND PWM_JOY_Jiao_R_DOWN1>10)THEN
		PWM_Y37_SET_Target:=800;  //开环  占控比   0-1000
	ELSE
		PWM_Y37_SET_Target:=0;
	END_IF
ELSE
	PWM_Y37_SET_Target:=0;
END_IF

IF((LeftMove_move OR RightMove_move)AND MainWinch_move)THEN
	PWM_Y1_Target:=REAL_TO_UINT(UINT_TO_REAL(PWM_JOY_JIAO)/1000*(PAR_Y2_PosFull-PAR_Y2_NegFull)+PAR_Y2_NegFull);
	PWM_Y2_Target:=0;
	PWM_Y37_SET_Target:=800;
END_IF*)
(*直线行走*)//Y2  Y40   行走阀
IF DIH_SA19 THEN
	PWM_Y37_SET_Target:=800;
	PWM_Y1_Target:=0;
ELSE
	PWM_Y37_SET_Target:=0;
END_IF

IF((LeftMove_move OR RightMove_move)AND MainWinch_move)THEN
	PWM_Y2_Target:=REAL_TO_UINT(UINT_TO_REAL(PWM_JOY_JIAO)/1000*(PAR_Y2_PosFull-PAR_Y2_NegFull)+PAR_Y2_NegFull);
	PWM_Y1_Target:=0;
	PWM_Y37_SET_Target:=800;
END_IF


RAMP21(
	IN:=UINT_TO_INT(PWM_Y37_SET_Target), 
	ASCEND:= R_RAMP_zhixian, 
	DESCEND:= F_RAMP_zhixian, 
	TIMEBASE:=TIMEBASE_zhixian , 
	RESET:=FALSE , 
	OUT=>UINT_TO_INT(PWM_Y37_SET));


IF(PWM_JOYX_R_UP<=500)THEN
	PWM_JOYX_R_UP_a:=PWM_JOYX_R_UP;
	PWM_JOYX_R_UP_b:=0;
ELSE
	PWM_JOYX_R_UP_a:=500;
	PWM_JOYX_R_UP_b:=PWM_JOYX_R_UP-500;
END_IF

IF(PWM_JOYX_R_DOWN<=500)THEN
	PWM_JOYX_R_DOWN_a:=PWM_JOYX_R_DOWN;
	PWM_JOYX_R_DOWN_b:=0;
ELSE
	PWM_JOYX_R_DOWN_a:=500;
	PWM_JOYX_R_DOWN_b:=PWM_JOYX_R_DOWN-500;
END_IF

	
(*单动力头动作*)
IF (NOT MainWinch_move) AND(PowerHead_move) AND(NOT DI_RHandle_SB6) THEN
	IF PWM_JOYX_R_UP>10 THEN//动力头反转
			PWM_Y1_Target:=REAL_TO_UINT(UINT_TO_REAL(PWM_JOYX_R_UP)/1000*(PAR_Y1_PosFull-PAR_Y1_NegFull)+PAR_Y1_NegFull);			
			PWM_Y2_Target:=REAL_TO_UINT(UINT_TO_REAL(PWM_JOYX_R_UP_b)/500*(PAR_Y2_PosFull-PAR_Y2_NegFull)+PAR_Y2_NegFull);
		IF(DIH_SA18)THEN
			PWM_Y1_Target:=0;			
			PWM_Y2_Target:=REAL_TO_UINT(UINT_TO_REAL(PWM_JOYX_R_UP)/1000*(PAR_Y2_PosFull-PAR_Y2_NegFull)+PAR_Y2_NegFull);
		END_IF
		PWM_Y12_SET_Tatget:=REAL_TO_UINT(UINT_TO_REAL(PWM_JOYX_R_UP)/1000*(PAR_Valve1_PosFull-PAR_Valve1_NegFull)+PAR_Valve1_NegFull);
		PWM_Y61_SET_Tatget:=REAL_TO_UINT(UINT_TO_REAL(PWM_JOYX_R_UP)/1000*(PAR_Valve1_PosFull-PAR_Valve1_NegFull)+PAR_Valve1_NegFull);
		PWM_Y14_SET_Tatget:=REAL_TO_UINT(UINT_TO_REAL(PWM_JOYX_R_UP_b)/500*(PAR_Valve2_PosFull-PAR_Valve2_NegFull)+PAR_Valve2_NegFull);
		PWM_Y11_SET:=0;
		PWM_Y13_SET:=0;
		PWM_Y60_SET:=0;
		PWM_Y11_SET_Tatget:=0;
		PWM_Y13_SET_Tatget:=0;
		PWM_Y60_SET_Tatget:=0;
		IF(PWM_JOYX_R_UP>700)THEN
			PWM_Y41_SET:=PAR_Valve2_PosFull;//快速回油阀
		END_IF
		PWM_Y59_SET:=0;
		PWM_Y42_SET:=0;
	ELSIF PWM_JOYX_R_DOWN>10 THEN //动力头正转
			PWM_Y1_Target:=REAL_TO_UINT(UINT_TO_REAL(PWM_JOYX_R_DOWN)/1000*(PAR_Y1_PosFull-PAR_Y1_NegFull)+PAR_Y1_NegFull);			
			PWM_Y2_Target:=REAL_TO_UINT(UINT_TO_REAL(PWM_JOYX_R_DOWN_b)/500*(PAR_Y2_PosFull-PAR_Y2_NegFull)+PAR_Y2_NegFull);
		IF(DIH_SA18)THEN
			PWM_Y1_Target:=0;			
			PWM_Y2_Target:=REAL_TO_UINT(UINT_TO_REAL(PWM_JOYX_R_DOWN)/1000*(PAR_Y2_PosFull-PAR_Y2_NegFull)+PAR_Y2_NegFull);
		END_IF
			PWM_Y11_SET_Tatget:=REAL_TO_UINT(UINT_TO_REAL(PWM_JOYX_R_DOWN)/1000*(PAR_Valve1_PosFull-PAR_Valve1_NegFull)+PAR_Valve1_NegFull);
			PWM_Y60_SET_Tatget:=REAL_TO_UINT(UINT_TO_REAL(PWM_JOYX_R_DOWN)/1000*(PAR_Valve1_PosFull-PAR_Valve1_NegFull)+PAR_Valve1_NegFull);		
			PWM_Y13_SET_Tatget:=REAL_TO_UINT(UINT_TO_REAL(PWM_JOYX_R_DOWN_b)/500*(PAR_Valve2_PosFull-PAR_Valve2_NegFull)+PAR_Valve2_NegFull);
		IF(PWM_JOYX_R_DOWN>700)THEN
		PWM_Y59_SET:=PAR_Valve2_PosFull;//合流
		PWM_Y42_SET:=PAR_Valve2_PosFull;//快速回油阀
		END_IF
		PWM_Y41_SET:=0;
		PWM_Y12_SET:=0;
		PWM_Y14_SET:=0;
		PWM_Y61_SET:=0;	
		PWM_Y12_SET_Tatget:=0;
		PWM_Y14_SET_Tatget:=0;
		PWM_Y61_SET_Tatget:=0;
	END_IF
ELSIF (MainWinch_move) AND(PowerHead_move) AND( NOT DI_RHandle_SB6) THEN
	//主卷和动力头复合动作时 主泵2提供给动力头油
	IF PWM_JOYX_R_UP>10 THEN//动力头反转 
		IF(PWM_JOYY_L_DOWN>10) THEN//主卷上提
		PWM_JOY_P:=MAX(PWM_JOYY_L_DOWN,PWM_JOYX_R_UP);
		PWM_Y1_Target:=REAL_TO_UINT(UINT_TO_REAL(PWM_JOY_P)/1000*(PAR_Y2_PosFull-PAR_Y2_NegFull)+PAR_Y2_NegFull);
		PWM_Y12_SET_Tatget:=REAL_TO_UINT(UINT_TO_REAL(PWM_JOYX_R_UP)/1000*(PAR_Valve2_PosFull-400)*P_value+400);
		PWM_Y11_SET_Tatget:=0;
		PWM_Y14_SET_Tatget:=0;
		PWM_Y13_SET_Tatget:=0;
		PWM_Y60_SET_Tatget:=0;
		PWM_Y61_SET_Tatget:=0;
		PWM_Y41_SET:=PAR_Valve2_PosFull;
		PWM_Y42_SET:=0;
		PWM_Y59_SET:=0;
		ELSIF PWM_JOYY_L_UP>10 THEN//主卷下放
 		PWM_Y1_Target:=REAL_TO_UINT(UINT_TO_REAL(PWM_JOYX_R_UP)/1000*(PAR_Y2_PosFull-PAR_Y2_NegFull)+PAR_Y2_NegFull);
		PWM_Y12_SET_Tatget:=REAL_TO_UINT(UINT_TO_REAL(PWM_JOYX_R_UP)/1000*(PAR_Valve2_PosFull-PAR_Valve2_NegFull)+PAR_Valve2_NegFull);
		PWM_Y11_SET_Tatget:=0;
		PWM_Y14_SET_Tatget:=0;
		PWM_Y13_SET_Tatget:=0;
		PWM_Y60_SET_Tatget:=0;
		PWM_Y61_SET_Tatget:=0;
		PWM_Y41_SET:=PAR_Valve2_PosFull;
		PWM_Y59_SET:=0;	
		PWM_Y42_SET:=0;
		END_IF
		
		
	ELSIF PWM_JOYX_R_DOWN>10 THEN //动力头正转
		PWM_Y1_Target:=REAL_TO_UINT(UINT_TO_REAL(PWM_JOYX_R_DOWN)/1000*(PAR_Y2_PosFull-PAR_Y2_NegFull)+PAR_Y2_NegFull);
		PWM_Y11_SET_Tatget:=REAL_TO_UINT(UINT_TO_REAL(PWM_JOYX_R_DOWN)/1000*(PAR_Valve2_PosFull-PAR_Valve2_NegFull)+PAR_Valve2_NegFull);
		PWM_Y13_SET_Tatget:=0;
		PWM_Y12_SET_Tatget:=0;
		PWM_Y14_SET_Tatget:=0;
		PWM_Y60_SET_Tatget:=0;
		PWM_Y61_SET_Tatget:=0;
		PWM_Y41_SET:=0;
		PWM_Y42_SET:=PAR_Valve2_PosFull;
		PWM_Y59_SET:=0;	
	END_IF	
ELSE
		PWM_Y12_SET_Tatget:=0;
		PWM_Y14_SET_Tatget:=0;
		PWM_Y61_SET_Tatget:=0;
		PWM_Y11_SET_Tatget:=0;
		PWM_Y13_SET_Tatget:=0;
		PWM_Y60_SET_Tatget:=0;
		PWM_Y41_SET:=0;
		PWM_Y42_SET:=0;	
		PWM_Y59_SET:=0;	
END_IF


//判断抛土模式
Rtrig_DongLiTou1(clk:=(CANI_JOYX_R>3000));//反转判断
IF Rtrig_DongLiTou1.Q THEN
	Count_TIMES_Fanzhuan:=Count_TIMES_Fanzhuan + 1;
END_IF
Rtrig_DongLiTou2(clk:=(CANI_JOYX_R<2000));//正转判断
IF Rtrig_DongLiTou2.Q THEN
	Count_TIMES_Zhengzhuan:=Count_TIMES_Zhengzhuan + 1;
END_IF	
IF (Count_TIMES_Fanzhuan_LAST<>Count_TIMES_Fanzhuan) AND (Count_TIMES_Zhengzhuan_LAST<>Count_TIMES_Zhengzhuan) THEN
	Paotu_Modle:=TRUE;
END_IF
TIME_1000ms(IN:=NOT TIME_1000ms.Q,PT:=T#800MS);
IF (TIME_1000ms.Q) THEN
	Count_TIMES_Fanzhuan_LAST:=Count_TIMES_Fanzhuan;
	Count_TIMES_Zhengzhuan_LAST:=Count_TIMES_Zhengzhuan;
END_IF

IF(Count_TIMES_Fanzhuan_LAST=Count_TIMES_Fanzhuan) AND (Count_TIMES_Zhengzhuan_LAST=Count_TIMES_Zhengzhuan) THEN
	PaoTU_biaozhi:=TRUE;
ELSE
	PaoTU_biaozhi:=FALSE;	
END_IF
TIME_1000ms_TP(IN:=PaoTU_biaozhi,PT:=T#800MS);
IF TIME_1000ms_TP.Q OR MainWinch_move  THEN
	Paotu_Modle:=FALSE;
END_IF

IF(NOT CANI_WorkModeSwitch) THEN
	Paotu_Modle:=FALSE;
END_IF

IF Paotu_Modle THEN
	TIMEBASE_ratate:=T#20MS;
ELSE
	TIMEBASE_ratate:=T#100MS;
END_IF


(*动力头动作缓冲*)
//启动缓冲时间300ms，停止缓冲时间600ms
(*动力头动作缓冲*)
//启动缓冲时间300ms，停止缓冲时间600ms
RAMP1(
	IN:=WORD_TO_INT(PWM_Y11_SET_Tatget), 
	ASCEND:= R_RAMP_ratate, 
	DESCEND:= F_RAMP_ratate, 
	TIMEBASE:=TIMEBASE_ratate , 
	RESET:=FALSE , 
	OUT=>(PWM_Y11_SET_Tatget1));
IF(PWM_Y11_SET_Tatget1>=400) THEN
	Curve_input:=TO_UINT(PWM_Y11_SET_Tatget1 - 400);
	IF(Curve_input>900) THEN
		Curve_input:=900;
	END_IF
	curve1(input:=REAL_TO_UINT(UINT_TO_REAL(Curve_input)*72.8),Zero:=FALSE,Full:=FALSE,
		   PAR_Progression:=Curve_Par,OutputEnable:=TRUE);
	PWM_Y11_SET:=PAR_Valve1_NegFull + REAL_TO_UINT(UINT_TO_REAL(curve1.Output)/72.8);
ELSE
	PWM_Y11_SET:=0;
END_IF

RAMP2(
	IN:=WORD_TO_INT(PWM_Y12_SET_Tatget), 
	ASCEND:= R_RAMP_ratate, 
	DESCEND:= F_RAMP_ratate, 
	TIMEBASE:=TIMEBASE_ratate , 
	RESET:=FALSE , 
	OUT=>(PWM_Y12_SET_Tatget1));
IF(PWM_Y12_SET_Tatget1>=400) THEN
	Curve_input:=TO_UINT(PWM_Y12_SET_Tatget1 - 400);
	IF(Curve_input>900) THEN
		Curve_input:=900;
	END_IF
	curve2(input:=REAL_TO_UINT(UINT_TO_REAL(Curve_input)*72.8),Zero:=FALSE,Full:=FALSE,
		   PAR_Progression:=Curve_Par,OutputEnable:=TRUE);
	PWM_Y12_SET:=PAR_Valve1_NegFull + REAL_TO_UINT(UINT_TO_REAL(curve2.Output)/72.8);
ELSE
	PWM_Y12_SET:=0;
END_IF

RAMP3(
	IN:=WORD_TO_INT(PWM_Y13_SET_Tatget), 
	ASCEND:= R_RAMP_ratate, 
	DESCEND:= F_RAMP_ratate, 
	TIMEBASE:=TIMEBASE_ratate , 
	RESET:=FALSE , 
	OUT=>(PWM_Y13_SET_Tatget1));
IF(PWM_Y13_SET_Tatget1>=400) THEN
	Curve_input:=TO_UINT(PWM_Y13_SET_Tatget1 - 400);
	IF(Curve_input>900) THEN
		Curve_input:=900;
	END_IF
	curve3(input:=REAL_TO_UINT(UINT_TO_REAL(Curve_input)*72.8),Zero:=FALSE,Full:=FALSE,
		   PAR_Progression:=Curve_Par,OutputEnable:=TRUE);
	PWM_Y13_SET:=PAR_Valve1_NegFull + REAL_TO_UINT(UINT_TO_REAL(curve3.Output)/72.8);
ELSE
	PWM_Y13_SET:=0;
END_IF

RAMP4(
	IN:=WORD_TO_INT(PWM_Y14_SET_Tatget), 
	ASCEND:= R_RAMP_ratate, 
	DESCEND:= F_RAMP_ratate, 
	TIMEBASE:=TIMEBASE_ratate , 
	RESET:=FALSE , 
	OUT=>(PWM_Y14_SET_Tatget1));
IF(PWM_Y14_SET_Tatget1>=400) THEN
	Curve_input:=TO_UINT(PWM_Y14_SET_Tatget1 - 400);
	IF(Curve_input>900) THEN
		Curve_input:=900;
	END_IF
	curve4(input:=REAL_TO_UINT(UINT_TO_REAL(Curve_input)*72.8),Zero:=FALSE,Full:=FALSE,
		   PAR_Progression:=Curve_Par,OutputEnable:=TRUE);
	PWM_Y14_SET:=PAR_Valve1_NegFull + REAL_TO_UINT(UINT_TO_REAL(curve4.Output)/72.8);
ELSE
	PWM_Y14_SET:=0;
END_IF

RAMP5(
	IN:=WORD_TO_INT(PWM_Y60_SET_Tatget), 
	ASCEND:= R_RAMP_ratate, 
	DESCEND:= F_RAMP_ratate, 
	TIMEBASE:=TIMEBASE_ratate , 
	RESET:=FALSE , 
	OUT=>(PWM_Y60_SET_Tatget1));
IF(PWM_Y60_SET_Tatget1>=400) THEN
	Curve_input:=TO_UINT(PWM_Y60_SET_Tatget1 - 400);
	IF(Curve_input>900) THEN
		Curve_input:=900;
	END_IF
	curve5(input:=REAL_TO_UINT(UINT_TO_REAL(Curve_input)*72.8),Zero:=FALSE,Full:=FALSE,
		   PAR_Progression:=Curve_Par,OutputEnable:=TRUE);
	PWM_Y60_SET:=PAR_Valve1_NegFull + REAL_TO_UINT(UINT_TO_REAL(curve5.Output)/72.8);
ELSE
	PWM_Y60_SET:=0;
END_IF

RAMP6(
	IN:=WORD_TO_INT(PWM_Y61_SET_Tatget), 
	ASCEND:= R_RAMP_ratate, 
	DESCEND:= F_RAMP_ratate, 
	TIMEBASE:=TIMEBASE_ratate , 
	RESET:=FALSE , 
	OUT=>(PWM_Y61_SET_Tatget1));
IF(PWM_Y61_SET_Tatget1>=400) THEN
	Curve_input:=TO_UINT(PWM_Y61_SET_Tatget1 - 400);
	IF(Curve_input>900) THEN
		Curve_input:=900;
	END_IF
	curve6(input:=REAL_TO_UINT(UINT_TO_REAL(Curve_input)*72.8),Zero:=FALSE,Full:=FALSE,
		   PAR_Progression:=Curve_Par,OutputEnable:=TRUE);
	PWM_Y61_SET:=PAR_Valve1_NegFull + REAL_TO_UINT(UINT_TO_REAL(curve6.Output)/72.8);
ELSE
	PWM_Y61_SET:=0;
END_IF


IF(PWM_Y5_SET>1300)THEN
	PWM_Y5_SET :=1300;
END_IF
IF(PWM_Y6_SET>1300)THEN
	PWM_Y6_SET :=1300;
END_IF
IF(PWM_Y15_SET>1300)THEN
	PWM_Y15_SET :=1300;
END_IF
IF(PWM_Y16_SET>1300)THEN
	PWM_Y16_SET :=1300;
END_IF	
IF(PWM_Y11_SET>1300)THEN
	PWM_Y11_SET :=1300;
END_IF
IF(PWM_Y12_SET>1300)THEN
	PWM_Y12_SET :=1300;
END_IF
IF(PWM_Y13_SET>1300)THEN
	PWM_Y13_SET :=1300;
END_IF
IF(PWM_Y14_SET>1300)THEN
	PWM_Y14_SET :=1300;
END_IF
IF(PWM_Y60_SET>1300)THEN
	PWM_Y60_SET :=1300;
END_IF
IF(PWM_Y61_SET>1300)THEN
	PWM_Y61_SET :=1300;
END_IF


IF(PWM_Y11_SET<=300)THEN
	PWM_Y11_SET :=0;
END_IF
IF(PWM_Y12_SET<=300)THEN
	PWM_Y12_SET :=0;
END_IF
IF(PWM_Y13_SET<=300)THEN
	PWM_Y13_SET :=0;
END_IF
IF(PWM_Y14_SET<=300)THEN
	PWM_Y14_SET :=0;
END_IF
IF(PWM_Y60_SET<=300)THEN
	PWM_Y60_SET :=0;
END_IF
IF(PWM_Y61_SET<=300)THEN
	PWM_Y61_SET :=0;
END_IF


BiaoZHI_MainWinchUp:=FALSE;
IF(PWM_JOYY_L_UP<=500)THEN
	PWM_JOYY_L_UP_a:=PWM_JOYY_L_UP;
	PWM_JOYY_L_UP_b:=0;
ELSE
	PWM_JOYY_L_UP_a:=500;
	PWM_JOYY_L_UP_b:=PWM_JOYY_L_UP-500;
END_IF

IF(PWM_JOYY_L_DOWN<=500)THEN
	PWM_JOYY_L_DOWN_a:=PWM_JOYY_L_DOWN;
	PWM_JOYY_L_DOWN_b:=0;
ELSE
	PWM_JOYY_L_DOWN_a:=500;
	PWM_JOYY_L_DOWN_b:=PWM_JOYY_L_DOWN-500;
END_IF



(*单主卷动作*)
IF ( MainWinch_move) AND (NOT PowerHead_move) AND (NOT LeftMove_move) AND (NOT RightMove_move)THEN
	IF PWM_JOYY_L_UP>10   THEN//主卷下放
		PWM_Y1_Target:=REAL_TO_UINT(UINT_TO_REAL(PWM_JOYY_L_UP)/1000*(PAR_Y1_PosFull-PAR_Y1_NegFull)+PAR_Y1_NegFull);
		PWM_Y2_Target:=REAL_TO_UINT(UINT_TO_REAL(PWM_JOYY_L_UP)/1000*(PAR_Y2_PosFull-PAR_Y2_NegFull)+PAR_Y2_NegFull);
		BiaoZHI_MainWinchUp:=TRUE;
		PWM_Y8_SET_Target:=REAL_TO_UINT(UINT_TO_REAL(PWM_JOYY_L_UP)/1000*(PAR_Valve1_PosFull-PAR_Valve1_NegFull)+PAR_Valve1_NegFull);
		PWM_Y10_SET_Target:=REAL_TO_UINT(UINT_TO_REAL(PWM_JOYY_L_UP)/1000*(PAR_Valve2_PosFull-PAR_Valve2_NegFull)+PAR_Valve2_NegFull);
		PWM_Y7_SET_Target:=0;
		PWM_Y9_SET_Target:=0;
		IF(DIH_SA19)THEN
			PWM_Y10_SET_Target:=0;
			PWM_Y9_SET_Target:=0;
			PWM_Y2_Target:=0;	
		END_IF
	ELSIF PWM_JOYY_L_DOWN>10 THEN//主卷上提
		PWM_Y1_Target:=REAL_TO_UINT(UINT_TO_REAL(PWM_JOYY_L_DOWN)/1000*(PAR_Y1_PosFull-PAR_Y1_NegFull)+PAR_Y1_NegFull);
		PWM_Y2_Target:=REAL_TO_UINT(UINT_TO_REAL(PWM_JOYY_L_DOWN)/1000*(PAR_Y2_PosFull-PAR_Y2_NegFull)+PAR_Y2_NegFull);
		PWM_Y7_SET_Target:=REAL_TO_UINT(UINT_TO_REAL(PWM_JOYY_L_DOWN)/1000*(PAR_Valve1_PosFull-PAR_Valve2_NegFull)+PAR_Valve2_NegFull);
		PWM_Y9_SET_Target:=REAL_TO_UINT(UINT_TO_REAL(PWM_JOYY_L_DOWN)/1000*(PAR_Valve2_PosFull-PAR_Valve2_NegFull)+PAR_Valve2_NegFull);
		PWM_Y8_SET_Target:=0;
		PWM_Y10_SET_Target:=0;	
		IF(DIH_SA19)THEN
			PWM_Y10_SET_Target:=0;
			PWM_Y9_SET_Target:=0;
			PWM_Y2_Target:=0;	
		END_IF
	END_IF
ELSIF( MainWinch_move) AND (PowerHead_move) THEN
	//主卷和动力头复合动作时 主泵1提供给主卷油
	IF PWM_JOYY_L_UP>10 THEN//主卷下放
		IF(PWM_JOYX_R_DOWN>10) THEN //动力头正转
			PWM_JOY_P4:=MAX(PWM_JOYY_L_UP,PWM_JOYX_R_DOWN);
			PWM_Y2_Target:=REAL_TO_UINT(UINT_TO_REAL(PWM_JOYY_L_UP)/1000*(PAR_Y1_PosFull-PAR_Y1_NegFull)+PAR_Y1_NegFull);
			PWM_Y1_Target:=REAL_TO_UINT(UINT_TO_REAL(PWM_JOYY_L_UP)/1000*(PAR_Y1_PosFull-PAR_Y1_NegFull)+PAR_Y1_NegFull);
			PWM_Y10_SET_Target:=REAL_TO_UINT(UINT_TO_REAL(PWM_JOYY_L_UP)/1000*(PAR_Valve1_PosFull-PAR_Valve1_NegFull)+PAR_Valve1_NegFull);
			PWM_Y8_SET_Target:=REAL_TO_UINT(UINT_TO_REAL(1000-PWM_JOYX_R_DOWN)/1000*(PAR_Valve1_PosFull-PAR_Valve1_NegFull)+PAR_Valve1_NegFull);
			PWM_Y7_SET_Target:=0;
			PWM_Y9_SET_Target:=0;
		ELSIF PWM_JOYX_R_UP>10 THEN//动力头反转
			PWM_JOY_P3:=MAX(PWM_JOYY_L_UP,PWM_JOYX_R_UP);
			PWM_Y2_Target:=REAL_TO_UINT(UINT_TO_REAL(PWM_JOYY_L_UP)/1000*(PAR_Y1_PosFull-PAR_Y1_NegFull)+PAR_Y1_NegFull);
			PWM_Y1_Target:=REAL_TO_UINT(UINT_TO_REAL(PWM_JOYY_L_UP)/1000*(PAR_Y1_PosFull-PAR_Y1_NegFull)+PAR_Y1_NegFull);
			PWM_Y10_SET_Target:=REAL_TO_UINT(UINT_TO_REAL(PWM_JOYY_L_UP)/1000*(PAR_Valve1_PosFull-PAR_Valve1_NegFull)+PAR_Valve1_NegFull);
			PWM_Y8_SET_Target:=REAL_TO_UINT(UINT_TO_REAL(1000-PWM_JOYX_R_UP)/1000*(PAR_Valve1_PosFull-PAR_Valve1_NegFull)+PAR_Valve1_NegFull);
			PWM_Y7_SET_Target:=0;
			PWM_Y9_SET_Target:=0;
		END_IF	
	ELSIF PWM_JOYY_L_DOWN>10 THEN//主卷上提
		IF(PWM_JOYX_R_DOWN>10) THEN //动力头正转
			PWM_JOY_P2:=MAX(PWM_JOYY_L_DOWN,PWM_JOYX_R_DOWN);
			PWM_Y2_Target:=REAL_TO_UINT(UINT_TO_REAL(PWM_JOYY_L_DOWN)/1000*(PAR_Y1_PosFull-PAR_Y1_NegFull)+PAR_Y1_NegFull);
			PWM_Y1_Target:=REAL_TO_UINT(UINT_TO_REAL(PWM_JOYY_L_DOWN)/1000*(PAR_Y1_PosFull-PAR_Y1_NegFull)+PAR_Y1_NegFull);
			PWM_Y9_SET_Target:=REAL_TO_UINT(UINT_TO_REAL(PWM_JOYY_L_DOWN)/1000*(PAR_Valve1_PosFull-750)+750);
			PWM_Y7_SET_Target:=REAL_TO_UINT(UINT_TO_REAL(PWM_JOYY_L_DOWN)/1000*(PAR_Valve1_PosFull-750)+750);
			PWM_Y8_SET_Target:=0;
			PWM_Y10_SET_Target:=0;
		ELSIF PWM_JOYX_R_UP>10 THEN//动力头反转
			PWM_JOY_P1:=MAX(PWM_JOYY_L_DOWN,PWM_JOYX_R_UP);
			PWM_Y1_Target:=REAL_TO_UINT(UINT_TO_REAL(PWM_JOYY_L_DOWN)/1000*(PAR_Y1_PosFull-PAR_Y1_NegFull)+PAR_Y1_NegFull);
			PWM_Y2_Target:=REAL_TO_UINT(UINT_TO_REAL(PWM_JOYY_L_DOWN)/1000*(PAR_Y2_PosFull-PAR_Y2_NegFull)+PAR_Y2_NegFull);
			PWM_Y7_SET_Target:=REAL_TO_UINT(UINT_TO_REAL(PWM_JOYY_L_DOWN)/1000*(PAR_Valve1_PosFull-750)+750);
			PWM_Y9_SET_Target:=REAL_TO_UINT(UINT_TO_REAL(PWM_JOYY_L_DOWN)/1000*(PAR_Valve2_PosFull-750)+750);
			PWM_Y8_SET_Target:=0;
			PWM_Y10_SET_Target:=0;
		END_IF
	END_IF
ELSIF (MainWinch_move) AND (LeftMove_move OR RightMove_move) THEN
//主卷和行走复合动作 主泵1提供给主卷油
	IF PWM_JOYY_L_UP>10 THEN//主卷下放
		PWM_Y1_Target:=REAL_TO_UINT(UINT_TO_REAL(PWM_JOYY_L_UP)/1000*(PAR_Y1_PosFull-PAR_Y1_NegFull)+PAR_Y1_NegFull);
		PWM_Y10_SET_Target:=0;
		PWM_Y8_SET_Target:=PAR_Valve1_PosFull;
		PWM_Y7_SET_Target:=0;
		PWM_Y9_SET_Target:=0;
	ELSIF PWM_JOYY_L_DOWN>10 THEN//主卷上提
		PWM_Y1_Target:=REAL_TO_UINT(UINT_TO_REAL(PWM_JOYY_L_DOWN)/1000*(PAR_Y1_PosFull-PAR_Y1_NegFull)+PAR_Y1_NegFull);
		PWM_Y9_SET_Target:=0;
		PWM_Y7_SET_Target:=PAR_Valve1_PosFull;
		PWM_Y8_SET_Target:=0;
		PWM_Y10_SET_Target:=0;		
		PWM_Y19_SET:=0;
		IF(DI_LHandle_SB4)THEN
			PWM_Y20_SET:=600;
		ELSE
			PWM_Y20_SET:=0;
		END_IF
	END_IF
ELSE
		PWM_Y8_SET:=0;
		PWM_Y10_SET:=0;
		PWM_Y7_SET:=0;
		PWM_Y9_SET:=0;
		PWM_Y8_SET_Target:=0;
		PWM_Y10_SET_Target:=0;
		PWM_Y7_SET_Target:=0;
		PWM_Y9_SET_Target:=0;
END_IF
	
	
//主卷扬根据阀的开关调整斜坡值	
	IF(PWM_Y8_SET<1000  AND  PWM_Y8_SET>=900)THEN    //主卷下放斜坡值
			F_RAMP_mainwinch_down:=200;
	ELSIF(PWM_Y8_SET<900)THEN
			F_RAMP_mainwinch_down:=100;
	ELSE
			F_RAMP_mainwinch_down:=200;
	END_IF
		
	IF(PWM_Y7_SET<1000  AND  PWM_Y7_SET>=900)THEN  //主卷上提斜坡值
			F_RAMP_mainwinch_down:=300;
	ELSIF(PWM_Y7_SET<900  )THEN
			F_RAMP_mainwinch_down:=200;
	ELSE
			F_RAMP_mainwinch_down:=400;
	END_IF
		
RAMP7(
	IN:=WORD_TO_INT(PWM_Y7_SET_Target), 
	ASCEND:= R_RAMP_mainwinch, 
	DESCEND:= F_RAMP_mainwinch_up, 
	TIMEBASE:=TIMEBASE_mainwinch , 
	RESET:=FALSE , 
	OUT=>(PWM_Y7_SET_Target1));
IF(PWM_Y7_SET_Target1>=400) THEN
	Curve_input:=TO_UINT(PWM_Y7_SET_Target1 - 400);
	IF(Curve_input>900) THEN
		Curve_input:=900;
	END_IF
	curve7(input:=REAL_TO_UINT(UINT_TO_REAL(Curve_input)*72.8),Zero:=FALSE,Full:=FALSE,
		   PAR_Progression:=Curve_Par,OutputEnable:=TRUE);
	PWM_Y7_SET:=PAR_Valve1_NegFull + REAL_TO_UINT(UINT_TO_REAL(curve7.Output)/72.8);
ELSE
	PWM_Y7_SET:=0;
END_IF


RAMP8(
	IN:=WORD_TO_INT(PWM_Y8_SET_Target), 
	ASCEND:= R_RAMP_mainwinch, 
	DESCEND:= F_RAMP_mainwinch_down, 
	TIMEBASE:=TIMEBASE_mainwinch , 
	RESET:=FALSE , 
	OUT=>(PWM_Y8_SET_Target1));
IF(PWM_Y8_SET_Target1>=400) THEN
	Curve_input:=TO_UINT(PWM_Y8_SET_Target1 - 400);
	IF(Curve_input>900) THEN
		Curve_input:=900;
	END_IF
	curve8(input:=REAL_TO_UINT(UINT_TO_REAL(Curve_input)*72.8),Zero:=FALSE,Full:=FALSE,
		   PAR_Progression:=Curve_Par,OutputEnable:=TRUE);
	PWM_Y8_SET:=PAR_Valve1_NegFull + REAL_TO_UINT(UINT_TO_REAL(curve8.Output)/72.8);
ELSE
	PWM_Y8_SET:=0;
END_IF


RAMP9(
	IN:=WORD_TO_INT(PWM_Y9_SET_Target), 
	ASCEND:= R_RAMP_mainwinch, 
	DESCEND:= F_RAMP_mainwinch_up, 
	TIMEBASE:=TIMEBASE_mainwinch , 
	RESET:=FALSE , 
	OUT=>(PWM_Y9_SET_Target1));
IF(PWM_Y9_SET_Target1>=400) THEN
	Curve_input:=TO_UINT(PWM_Y9_SET_Target1 - 400);
	IF(Curve_input>900) THEN
		Curve_input:=900;
	END_IF
	curve9(input:=REAL_TO_UINT(UINT_TO_REAL(Curve_input)*72.8),Zero:=FALSE,Full:=FALSE,
		   PAR_Progression:=Curve_Par,OutputEnable:=TRUE);
	PWM_Y9_SET:=PAR_Valve1_NegFull + REAL_TO_UINT(UINT_TO_REAL(curve9.Output)/72.8);
ELSE
	PWM_Y9_SET:=0;
END_IF

RAMP10(
	IN:=WORD_TO_INT(PWM_Y10_SET_Target), 
	ASCEND:= R_RAMP_mainwinch, 
	DESCEND:= F_RAMP_mainwinch_down, 
	TIMEBASE:=TIMEBASE_mainwinch , 
	RESET:=FALSE , 
	OUT=>(PWM_Y10_SET_Target1));
IF(PWM_Y10_SET_Target1>=400) THEN
	Curve_input:=TO_UINT(PWM_Y10_SET_Target1 - 400);
	IF(Curve_input>900) THEN
		Curve_input:=900;
	END_IF
	curve10(input:=REAL_TO_UINT(UINT_TO_REAL(Curve_input)*72.8),Zero:=FALSE,Full:=FALSE,
		   PAR_Progression:=Curve_Par,OutputEnable:=TRUE);
	PWM_Y10_SET:=PAR_Valve1_NegFull + REAL_TO_UINT(UINT_TO_REAL(curve10.Output)/72.8);
ELSE
	PWM_Y10_SET:=0;
END_IF


IF(PWM_Y7_SET>1300)THEN
	PWM_Y7_SET :=1300;
END_IF
IF(PWM_Y8_SET>1300)THEN
	PWM_Y8_SET :=1300;
END_IF
IF(PWM_Y9_SET>1300)THEN
	PWM_Y9_SET :=1300;
END_IF
IF(PWM_Y10_SET>1300)THEN
	PWM_Y10_SET :=1300;
END_IF

IF(PWM_Y7_SET<=300)THEN
	PWM_Y7_SET :=0;
END_IF
IF(PWM_Y8_SET<=300)THEN
	PWM_Y8_SET :=0;
END_IF
IF(PWM_Y9_SET<=300)THEN
	PWM_Y9_SET :=0;
END_IF
IF(PWM_Y10_SET<=300)THEN
	PWM_Y10_SET :=0;
END_IF




(*主泵卸荷阀控制*)
		PWM_Y39_SET_Target:=MAX(PWM_Y8_SET_Target,PWM_Y7_SET_Target,PWM_Y12_SET_Tatget,PWM_Y11_SET_Tatget,PWM_Y3_SET,PWM_Y4_SET,PWM_Y15_SET_Target,PWM_Y16_SET_Target);
		PWM_Y40_SET_Target:=MAX(PWM_Y9_SET_Target,PWM_Y10_SET_Target,PWM_Y13_SET_Tatget,PWM_Y14_SET_Tatget,PWM_Y5_SET_Target,PWM_Y6_SET_Target,PWM_Y17_SET2,PWM_Y18_SET);
	(*卸荷动作缓冲*)
RAMP19(
	IN:=WORD_TO_INT(PWM_Y39_SET_Target), 
	ASCEND:= R_RAMP_xiehe, 
	DESCEND:= F_RAMP_xiehe, 
	TIMEBASE:=TIMEBASE_xiehe , 
	RESET:=FALSE , 
	OUT=>(PWM_Y39_SET_Target1));
IF(PWM_Y39_SET_Target1>=400) THEN
	Curve_input:=TO_UINT(PWM_Y39_SET_Target1 - 400);
	IF(Curve_input>900) THEN
		Curve_input:=900;
	END_IF
	curve19(input:=REAL_TO_UINT(UINT_TO_REAL(Curve_input)*72.8),Zero:=FALSE,Full:=FALSE,
		   PAR_Progression:=Curve_Par1,OutputEnable:=TRUE);
	PWM_Y39_SET:=PAR_Valve1_NegFull + REAL_TO_UINT(UINT_TO_REAL(curve19.Output)/72.8);
ELSE
	PWM_Y39_SET:=0;
END_IF


RAMP20(
	IN:=WORD_TO_INT(PWM_Y40_SET_Target), 
	ASCEND:= R_RAMP_xiehe, 
	DESCEND:= F_RAMP_xiehe, 
	TIMEBASE:=TIMEBASE_xiehe , 
	RESET:=FALSE , 
	OUT=>(PWM_Y40_SET_Target1));
IF(PWM_Y40_SET_Target1>=400) THEN
	Curve_input:=TO_UINT(PWM_Y40_SET_Target1 - 400);
	IF(Curve_input>900) THEN
		Curve_input:=900;
	END_IF
	curve20(input:=REAL_TO_UINT(UINT_TO_REAL(Curve_input)*72.8),Zero:=FALSE,Full:=FALSE,
		   PAR_Progression:=Curve_Par1,OutputEnable:=TRUE);
	PWM_Y40_SET:=PAR_Valve1_NegFull + REAL_TO_UINT(UINT_TO_REAL(curve20.Output)/72.8);
ELSE
	PWM_Y40_SET:=0;
END_IF

	//在行走时一个泵供油时,需要关闭另外一个 泵的起压阀
	IF PWM_Y37_SET>500 AND (NOT MainWinch_move) THEN
		PWM_Y39_SET:=0;
	END_IF
	
IF(PWM_Y39_SET>1300)THEN
	PWM_Y39_SET :=1300;
END_IF
IF(PWM_Y40_SET>1300)THEN
	PWM_Y40_SET :=1300;
END_IF

IF(PWM_Y39_SET<=300)THEN
	PWM_Y39_SET :=0;
END_IF
IF(PWM_Y40_SET<=300)THEN
	PWM_Y40_SET :=0;
END_IF

(*副卷扬动作*)
IF(ViceWinch_move)THEN
	IF PWM_JOYY_R_UP>10 THEN//副卷下放
		PWM_Y4_SET:=REAL_TO_UINT(UINT_TO_REAL(PWM_JOYY_R_UP)/1000*(1200-500)+500);
		PWM_Y3_SET:=0;
		IF(NOT MainWinch_move) OR (NOT PowerHead_move) THEN
			PWM_Y1_Target:=REAL_TO_UINT(UINT_TO_REAL(PWM_JOYY_R_UP)/1000*(PAR_KP-PAR_Y1_NegFull)+PAR_Y1_NegFull);
		END_IF
		
	ELSIF PWM_JOYY_R_DOWN>10 THEN//副卷上提
		PWM_Y3_SET:=REAL_TO_UINT(UINT_TO_REAL(PWM_JOYY_R_DOWN)/1000*(1200-500)+500);
		PWM_Y4_SET:=0;
		IF(NOT MainWinch_move) OR (NOT PowerHead_move) THEN
			PWM_Y1_Target:=REAL_TO_UINT(UINT_TO_REAL(PWM_JOYY_R_DOWN)/1000*(PAR_KP-PAR_Y1_NegFull)+PAR_Y1_NegFull);
		END_IF		
	END_IF
ELSE
	PWM_Y3_SET:=0;
	PWM_Y4_SET:=0;
END_IF

(*回转动作*)
//回转限制
IF  (CANO_DEPTH>980 AND  CANI_WorkModeSwitch) THEN
		Rotation_move:=FALSE;
END_IF
	
IF NOT DI_LHandle_SB7 THEN(*自动回转*) 
	IF  Rotation_move  OR DI_LHandle_SB2  THEN
		DOH_Y50_1 := TRUE;
		IF PWM_JOYX_L_UP>10 THEN// 右回转
			PWM_Y22_SET:=REAL_TO_UINT(UINT_TO_REAL(PWM_JOYX_L_UP)/1000*(PAR_ValveC_NegFull-PAR_Valve3_NegFull)+PAR_Valve3_NegFull);
			PWM_Y21_SET:=0;
		ELSIF PWM_JOYX_L_DOWN>10 THEN//左回转
			PWM_Y21_SET:=REAL_TO_UINT(UINT_TO_REAL(PWM_JOYX_L_DOWN)/1000*(PAR_ValveC_NegFull-PAR_Valve3_NegFull)+PAR_Valve3_NegFull);
			PWM_Y22_SET:=0;
		END_IF
	ELSE
		DOH_Y50_1:= FALSE;
		PWM_Y21_SET:=0;
		PWM_Y22_SET:=0;
	END_IF
ELSE
	DOH_Y50_1 := TRUE;
	IF(AUTO_ROTATION_VALVE>=0) THEN
		PWM_Y21_SET:=REAL_TO_UINT(INT_TO_REAL(ABS(AUTO_ROTATION_VALVE))*0.13);
	ELSE
		PWM_Y22_SET:=REAL_TO_UINT(INT_TO_REAL(ABS(AUTO_ROTATION_VALVE))*0.13);		
	END_IF
END_IF

//回转时警示灯响并且监控显示后界面
IF Rotation_move  OR DOH_Y50 THEN
	DOH_70:=TRUE;
	DOH_73:=TRUE;
	DOH_JK2:=TRUE;
ELSE
	DOH_70:=FALSE;
	DOH_73:=FALSE;
	DOH_JK2:=FALSE;
END_IF

//制动阀延时锁车
Rotation_late(IN:=DOH_Y50_1,PT:=T#2S);
IF  DOH_Y50_1 THEN
	DOH_Y50:=TRUE;
ELSE
	DOH_Y50:=Rotation_late.Q;
END_IF

(*加压动作*)
IF JiaYa_move THEN
	IF PWM_JOYY_R_UP>10 THEN//加压下
		PWM_Y23_SET_Taget:=REAL_TO_UINT(UINT_TO_REAL(PWM_JOYY_R_UP)/1000*(800-PAR_Valve3_NegFull)+PAR_Valve3_NegFull);
		PWM_Y24_SET_Taget:=0;
		
		IF(CANI_JiaYaFastSwitch OR DI_RHandle_SB7)THEN //加压快
			PWM_Y2_Target:=REAL_TO_UINT(UINT_TO_REAL(PWM_JOYY_R_UP)/1000*(500-300)+300);
			PWM_Y17_SET:=0;
			PWM_Y17_SET2:=0;
			PWM_Y18_SET_Taget:=1300;
		ELSE
			PWM_Y18_SET_Taget:=0;
		END_IF
		
	ELSIF PWM_JOYY_R_DOWN>10 THEN//加压上
		PWM_Y24_SET_Taget:=REAL_TO_UINT(UINT_TO_REAL(PWM_JOYY_R_DOWN)/1000*(800-PAR_Valve3_NegFull)+PAR_Valve3_NegFull);
		PWM_Y23_SET_Taget:=0;
		
		IF(CANI_JiaYaFastSwitch OR DI_RHandle_SB7)THEN //加压快
			PWM_Y2_Target:=REAL_TO_UINT(UINT_TO_REAL(PWM_JOYY_R_DOWN)/1000*(500-300)+300);
			PWM_Y17_SET:=800;
			PWM_Y17_SET2:=1300;
			PWM_Y18_SET:=0;
		ELSE
			PWM_Y18_SET:=0;
		END_IF
	END_IF
ELSE
	PWM_Y23_SET_Taget:=0;
	PWM_Y24_SET_Taget:=0;
	PWM_Y17_SET:=0;
	PWM_Y18_SET:=0;
	PWM_Y17_SET2:=0;
END_IF

RAMP22(
	IN:=WORD_TO_INT(PWM_Y23_SET_Taget), 
	ASCEND:= ASCEND_value, 
	DESCEND:= 5000, 
	TIMEBASE:=T#1000MS , 
	RESET:=FALSE , 
	OUT=>(PWM_Y23_SET_Taget1));
IF(PWM_Y23_SET_Taget1<310)THEN
		ASCEND_value:=6000;
ELSIF(PWM_Y23_SET_Taget1>=310 AND PWM_Y23_SET_Taget1<450)THEN
		ASCEND_value:=100;
ELSE
		ASCEND_value:=300;
END_IF
IF(PWM_Y23_SET_Taget1>=300) THEN
	Curve_input:=TO_UINT(PWM_Y23_SET_Taget1 - 300);
	IF(Curve_input>500) THEN
		Curve_input:=500;
	END_IF
	PWM_Y23_SET:=300 + Curve_input;
ELSE
	PWM_Y23_SET:=0;
END_IF

RAMP24(
	IN:=WORD_TO_INT(PWM_Y24_SET_Taget), 
	ASCEND:= 500, 
	DESCEND:= 500, //500-6000
	TIMEBASE:=T#300MS , 
	RESET:=FALSE , 
	OUT=>UINT_TO_INT(PWM_Y24_SET));
(*IF(PWM_Y24_SET_Taget1>=300) THEN
	Curve_input:=TO_UINT(PWM_Y24_SET_Taget1 - 300);
	IF(Curve_input>500) THEN
		Curve_input:=500;
	END_IF
	PWM_Y24_SET:=300 + Curve_input;
ELSE
	PWM_Y24_SET:=0;
END_IF*)



RAMP23(
	IN:=WORD_TO_INT(PWM_Y18_SET_Taget), 
	ASCEND:= ASCEND_value2, 
	DESCEND:= 5000, 
	TIMEBASE:=T#1000MS , 
	RESET:=FALSE , 
	OUT=>(PWM_Y18_SET_Taget1));
IF(PWM_Y18_SET_Taget1<610)THEN
		ASCEND_value2:=6000;
ELSE
	ASCEND_value2:=150;
END_IF	

IF(PWM_Y18_SET_Taget1>=600) THEN
	Curve_input:=TO_UINT(PWM_Y18_SET_Taget1 - 600);
	IF(Curve_input>700) THEN
		Curve_input:=700;
	END_IF
	PWM_Y18_SET:=600 + Curve_input;
ELSE
	PWM_Y18_SET:=0;
END_IF

(*PWM_Y23_SET:=PWM_Y23_SET_Taget;*)
IF JiaYa_move THEN
	IF PWM_JOYY_R_DOWN>10 THEN
		PWM_Y23_SET_Taget:=0;
		PWM_Y23_SET_Taget1:=0;
		PWM_Y23_SET:=0;
		PWM_Y18_SET_Taget1:=0;
		PWM_Y18_SET_Taget:=0;
		PWM_Y18_SET:=0;
	END_IF
END_IF

//加压限压
IF(CANI_DongLiTouPressLimitSwitch)THEN
	PWM_Y63_SET:=PAR_ValveD_PosFull;
ELSE
	PWM_Y63_SET:=0;
END_IF
		
(*平举动作*)
IF  BianFu_move THEN
	IF PWM_JOYY_R_UP>10 THEN//变幅下
		PWM_Y25_SET:=REAL_TO_UINT(UINT_TO_REAL(PWM_JOYY_R_UP)/1000*(PAR_Valve3_PosFull-PAR_Valve3_NegFull)+PAR_Valve3_NegFull);
		PWM_Y26_SET:=0;
	ELSIF PWM_JOYY_R_DOWN>10 THEN//变幅上
		PWM_Y26_SET:=REAL_TO_UINT(UINT_TO_REAL(PWM_JOYY_R_DOWN)/1000*(PAR_Valve3_PosFull-PAR_Valve3_NegFull)+PAR_Valve3_NegFull);
		PWM_Y25_SET:=0;
	END_IF
ELSE
	PWM_Y25_SET:=0;
	PWM_Y26_SET:=0;
END_IF

(*张紧等切换油缸动作*)
IF  LvZhang_move THEN
	IF(NOT CANI_LvDaiShenSuoSwitch)THEN
		IF PWM_JOYX_R_UP>10 THEN
			PWM_Y31_SET:=REAL_TO_UINT(UINT_TO_REAL(PWM_JOYX_R_UP)/1000*(PAR_Valve3_PosFull-PAR_Valve3_NegFull)+PAR_Valve3_NegFull);
			PWM_Y32_SET:=0;
			PWM_Y19_SET:=0;
			PWM_Y20_SET:=0;
		ELSIF PWM_JOYX_R_DOWN>10 THEN
			PWM_Y32_SET:=REAL_TO_UINT(UINT_TO_REAL(PWM_JOYX_R_DOWN)/1000*(PAR_Valve3_PosFull-PAR_Valve3_NegFull)+PAR_Valve3_NegFull);
			PWM_Y31_SET:=0;
			PWM_Y19_SET:=0;
			PWM_Y20_SET:=0;
		ELSE
			PWM_Y31_SET:=0;
			PWM_Y32_SET:=0;
			PWM_Y19_SET:=0;
			PWM_Y20_SET:=0;
		END_IF
	ELSE
		IF PWM_JOYX_R_UP>10 THEN
			PWM_Y19_SET:=REAL_TO_UINT(UINT_TO_REAL(PWM_JOYX_R_UP)/1000*(PAR_Valve3_PosFull-PAR_Valve3_NegFull)+PAR_Valve3_NegFull);
			PWM_Y20_SET:=0;
			PWM_Y31_SET:=0;
			PWM_Y32_SET:=0;
		ELSIF PWM_JOYX_R_DOWN>10 THEN
			PWM_Y20_SET:=REAL_TO_UINT(UINT_TO_REAL(PWM_JOYX_R_DOWN)/1000*(PAR_Valve3_PosFull-PAR_Valve3_NegFull)+PAR_Valve3_NegFull);
			PWM_Y19_SET:=0;
			PWM_Y31_SET:=0;
			PWM_Y32_SET:=0;
		ELSE
			PWM_Y31_SET:=0;
			PWM_Y32_SET:=0;
			PWM_Y19_SET:=0;
			PWM_Y20_SET:=0;
		END_IF
	END_IF
ELSE
	PWM_Y31_SET:=0;
	PWM_Y32_SET:=0;
	PWM_Y19_SET:=0;
	PWM_Y20_SET:=0;
END_IF


IF(CANI_ETouYouGangSwitch) THEN//支腿/鹅头油缸切换
	DOH_Y52:=TRUE;
ELSE
	DOH_Y52:=FALSE;
END_IF

//主卷动作及浮动时开锁
IF  MainWinch_move OR DOH_Y55 THEN
	DOH_Y53 := TRUE;
	DOH_Y64:=TRUE;
	GVL_SaveEngine.Y74:=TRUE;
ELSE
	DOH_Y53 := FALSE;	
	DOH_Y64:=FALSE;
	GVL_SaveEngine.Y74:=FALSE;
END_IF

(*主泵功率控制20230706*)
//区分发动机转速
MainPump_Pressure_Taget1450:=PAR_NegFull_x;
MainPump_Pressure_Taget1600:=PAR_PosFull_x;
MainPump_Pressure_Taget1750:=PAR_Zero_x;

IF EngineSpeedTarget<=1080 THEN SPEED_CASE:=1;
ELSIF EngineSpeedTarget>1080 AND EngineSpeedTarget<=1300 THEN SPEED_CASE:=2;
ELSIF EngineSpeedTarget>1300 AND EngineSpeedTarget<=1520 THEN SPEED_CASE:=3;
ELSIF EngineSpeedTarget>1520 AND EngineSpeedTarget<=1680 THEN SPEED_CASE:=4;
ELSIF EngineSpeedTarget>1680 AND EngineSpeedTarget<=1820 THEN SPEED_CASE:=5;
ELSIF EngineSpeedTarget>1820 THEN SPEED_CASE:=6;;END_IF
//不同转速下的发动机最大功率
CASE SPEED_CASE OF
1:  Enginer_Power:=135;
2:  Enginer_Power:=174;
3:  Enginer_Power:=200;
4:  Enginer_Power:=230;
5:  Enginer_Power:=250;
6:  Enginer_Power:=261;
END_CASE
//不同转速下的压力值
IF(CANO_Fubeng_Press>100)THEN
	CASE SPEED_CASE OF
		1:MainPump_Pressure_Taget:=MainPump_Pressure_Taget1000-HELIU_Press_Target1000;
		2:MainPump_Pressure_Taget:=MainPump_Pressure_Taget1200-HELIU_Press_Target1200;
		3:MainPump_Pressure_Taget:=MainPump_Pressure_Taget1450-HELIU_Press_Target1400;
		4:MainPump_Pressure_Taget:=MainPump_Pressure_Taget1600-HELIU_Press_Target1600;
		5:MainPump_Pressure_Taget:=MainPump_Pressure_Taget1750-HELIU_Press_Target1800;
		6:MainPump_Pressure_Taget:=MainPump_Pressure_Taget1900-HELIU_Press_Target1900;
	END_CASE
ELSE
	CASE SPEED_CASE OF
		1:MainPump_Pressure_Taget:=MainPump_Pressure_Taget1000;
		2:MainPump_Pressure_Taget:=MainPump_Pressure_Taget1200;
		3:MainPump_Pressure_Taget:=MainPump_Pressure_Taget1450;
		4:MainPump_Pressure_Taget:=MainPump_Pressure_Taget1600;
		5:MainPump_Pressure_Taget:=MainPump_Pressure_Taget1750;
		6:MainPump_Pressure_Taget:=MainPump_Pressure_Taget1900;
	END_CASE		
END_IF
IF( CANI_ECOSwitch) THEN
	CASE SPEED_CASE OF
		1:MainPump_Pressure_Taget:=MainPump_Pressure_Taget1000-ECO_Press_Target1000;
		2:MainPump_Pressure_Taget:=MainPump_Pressure_Taget1200-ECO_Press_Target1200;
		3:MainPump_Pressure_Taget:=MainPump_Pressure_Taget1450-ECO_Press_Target1400;
		4:MainPump_Pressure_Taget:=MainPump_Pressure_Taget1600-ECO_Press_Target1600;
		5:MainPump_Pressure_Taget:=MainPump_Pressure_Taget1750-ECO_Press_Target1800;
		6:MainPump_Pressure_Taget:=MainPump_Pressure_Taget1900-ECO_Press_Target1900;
	END_CASE
END_IF
MainPump_Pressure:=CANO_MainPUMP_Press1+CANO_MainPUMP_Press2;
//消除滤波
MainPump_Pressure_Subtract:= UINT_TO_INT(MainPump_Pressure-MainPump_Pressure_last1);

TIME_200ms(IN:=NOT TIME_200ms.Q,PT:=T#400MS);

IF(TIME_200ms.Q)THEN
	CANI_JOYX_R_last:=CANI_JOYX_R;
END_IF
Sub_Joyx_r:=UINT_TO_INT(CANI_JOYX_R_last) - UINT_TO_INT(CANI_JOYX_R);
IF(Sub_Joyx_r<-1200 OR Sub_Joyx_r>1200) THEN
	Joyx_change_bool:=TRUE;
	
END_IF

IF(CANI_JOYX_R=2500)THEN
	tempbool:=TRUE;
ELSE
	tempbool:=FALSE;
END_IF

TIME_1000_1ms(in:=tempbool,PT:=T#500MS);
IF(TIME_1000_1ms.Q)THEN
	JOY_PAOTU:=FALSE;
END_IF

TIME_400ms(IN:=Joyx_change_bool,PT:=T#10MS);
IF(TIME_400ms.Q) THEN
	Joyx_change_bool:=FALSE;
END_IF



//大范围波动
IF MainPump_Pressure_Subtract>270 OR MainPump_Pressure_Subtract<-270 THEN
	Subtract:=TRUE;
ELSE
	Subtract:=FALSE;	
END_IF
	TIME_LvBo4(IN:=Subtract,PT:=T#10MS);
	
IF(TIME_LvBo4.Q) AND (CANO_MainPUMP_Press1>210) THEN 
		MainPump_Pressure_ChangeBool1:=TRUE;
END_IF
	TIME_LvBo1(IN:=MainPump_Pressure_ChangeBool1,PT:=T#2S);
IF(TIME_LvBo1.Q) THEN
	MainPump_Pressure_ChangeBool1 :=FALSE;
END_IF

IF(MainPump_Pressure_ChangeBool1) AND (MainPump_Pressure>MainPump_Pressure_last1) THEN 
	MainPump_Pressure_last1:=MainPump_Pressure;
END_IF

//小范围波动
t_powertime:=TO_TIME(PAR_DeadBand_x);
IF (NOT MainPump_Pressure_ChangeBool1) THEN
	IF(MainPump_Pressure_Subtract>40 OR MainPump_Pressure_Subtract<-40)THEN 
		MainPump_Pressure_ChangeBool:=TRUE;
	ELSE
		MainPump_Pressure_ChangeBool:=FALSE;
	END_IF

	TIME_LvBo2(IN:=MainPump_Pressure_ChangeBool,PT:=t_powertime);
	IF(TIME_LvBo2.Q )THEN
		MainPump_Pressure_last1:=MainPump_Pressure;
	END_IF	
END_IF


IF PowerHead_move AND NOT(MainWinch_move) THEN
		JianGE2:=0.005;
ELSE
	IF(EngineSpeedTarget>1000 AND EngineSpeedTarget<1300)THEN
		JianGE2:=0.005;
	ELSE
		JianGE2:=0.005;
	END_IF
END_IF
	
IF MainPump_Pressure_last1>MainPump_Pressure_Taget THEN
	Pressure_Coe_Taget:=UINT_TO_REAL(MainPump_Pressure_Taget)/UINT_TO_REAL(MainPump_Pressure_last1);(*压力系数*)
ELSE
	Pressure_Coe_Taget:=1;
END_IF
Pressure_Coe := Pressure_Coe_Taget;


IF MainPump_Pressure_last1>MainPump_Pressure_Taget  THEN
	IF(PWM_Y1_Target>=PAR_Y1_1_NegFull)THEN
		PWM_Y1_Target_OutPut:=REAL_TO_UINT(UINT_TO_REAL(PWM_Y1_Target-PAR_Y1_1_NegFull)*Pressure_Coe+PAR_Y1_1_NegFull);
	END_IF
	IF(PWM_Y2_Target>=PAR_Y1_1_NegFull)THEN
		PWM_Y2_Target_OutPut:=REAL_TO_UINT(UINT_TO_REAL(PWM_Y2_Target-PAR_Y1_1_NegFull)*Pressure_Coe+PAR_Y1_1_NegFull);
	END_IF
ELSE
	PWM_Y1_Target_OutPut:=PWM_Y1_Target;
	PWM_Y2_Target_OutPut:=PWM_Y2_Target;
END_IF

IF(EngineSpeedTarget>CANO_SPEED AND CANO_SPEED>400)THEN
	EngineSpeedSub:=EngineSpeedTarget - CANO_SPEED;
ELSE
	EngineSpeedSub:=0;
END_IF

IF(PWM_Y1_Target_OutPut<300)THEN PWM_Y1_Target_OutPut:=300;END_IF	
IF(PWM_Y2_Target_OutPut<300)THEN PWM_Y2_Target_OutPut:=300;END_IF

RAMP15_IN:=PWM_Y1_Target_OutPut;
RAMP16_IN:=PWM_Y2_Target_OutPut;


IF MainWinch_move  OR  LeftMove_move OR RightMove_move THEN  
	TIMEBASE_pump:=T#1000MS;
	TIMEBASE_xiehe:=T#500MS;
ELSE
	TIMEBASE_pump:=T#600MS;
	TIMEBASE_xiehe:=T#300MS;
END_IF
t_PowerHead_move(IN:= MainWinch_move,PT:=T#4S);
IF t_PowerHead_move.Q THEN
	F_RAMP_pump:=x_t_PowerHead_move;
	R_RAMP_pump:=x2_t_PowerHead_move;
ELSE
       CASE SPEED_CASE OF
                1:F_RAMP_pump:=1500; R_RAMP_pump:=100;                  
                2: 		IF MainWinch_move AND (JiaYa_move OR CANO_JiayaPressure>80)  THEN    //3泵同时起压时，降低主泵的加载速度，避免掉速熄火
                                F_RAMP_pump:=1500; R_RAMP_pump:=100;
                        ELSE
                                F_RAMP_pump:=1500; R_RAMP_pump:=100;//从200降
                                IF  PWM_JOYY_L_UP>10 THEN
                                 F_RAMP_pump:=1500; R_RAMP_pump:=200;
                                END_IF
                        END_IF            
                3:
                        IF MainWinch_move AND (JiaYa_move OR CANO_JiayaPressure>80)  THEN    //3泵同时起压时，降低主泵的加载速度，避免掉速熄火
                                F_RAMP_pump:=1500; R_RAMP_pump:=150;
                        ELSE
                                F_RAMP_pump:=1500; R_RAMP_pump:=TO_INT(PAR_NegFull_y);
                                IF  PWM_JOYY_L_UP>10 THEN
                                 F_RAMP_pump:=1500; R_RAMP_pump:=300;
                                END_IF
                        END_IF                
                4:
                        IF MainWinch_move AND (JiaYa_move OR CANO_JiayaPressure>80)  THEN
                                F_RAMP_pump:=1500; R_RAMP_pump:=150;
                        ELSE
                                F_RAMP_pump:=1500; R_RAMP_pump:=TO_INT(PAR_PosFull_y);//从200降
                                IF  PWM_JOYY_L_UP>10 THEN
                                 F_RAMP_pump:=1500; R_RAMP_pump:=300;
                                END_IF
                        END_IF                                
                5:
                        IF MainWinch_move AND (JiaYa_move OR CANO_JiayaPressure>80)  THEN
                                F_RAMP_pump:=1500; R_RAMP_pump:=200;
                        ELSE
                                F_RAMP_pump:=1500; R_RAMP_pump:=TO_INT(PAR_Zero_y);
                                IF  PWM_JOYY_L_UP>10 THEN
                                 F_RAMP_pump:=1500; R_RAMP_pump:=300;
                                END_IF
                        END_IF                        
                6:		IF MainWinch_move AND (JiaYa_move OR CANO_JiayaPressure>80)  THEN
                                F_RAMP_pump:=1500; R_RAMP_pump:=200;
                        ELSE
                                F_RAMP_pump:=1500; R_RAMP_pump:=200;
                                IF  PWM_JOYY_L_UP>10 THEN
                                 F_RAMP_pump:=1500; R_RAMP_pump:=300;
                                END_IF
                        END_IF               
         END_CASE	
END_IF

RAMP15(
	IN:=UINT_TO_INT(RAMP15_IN), 
	ASCEND:= R_RAMP_pump, 
	DESCEND:= F_RAMP_pump, 
	TIMEBASE:=TIMEBASE_pump , 
	RESET:=FALSE , 
	OUT=>(PWM_Y1_SET));
	
RAMP16(
	IN:=UINT_TO_INT(RAMP16_IN), 
	ASCEND:= R_RAMP_pump, 
	DESCEND:= F_RAMP_pump, 
	TIMEBASE:=TIMEBASE_pump , 
	RESET:=FALSE , 
	OUT=>(PWM_Y2_SET));

IF (NOT Rotation_move) AND (NOT MainWinch_move) AND (NOT PowerHead_move)
		AND (NOT JiaYa_move) AND (NOT ViceWinch_move)
		AND (NOT LeftMove_move) AND (NOT RightMove_move)  THEN
	PWM_Y1_Target:=0;
	PWM_Y2_Target:=0;
END_IF


IF PWM_Y1_SET<TO_INT(PAR_Y1_1_NegFull )THEN
	PWM_Y1_SET:=TO_INT(PAR_Y1_1_NegFull);
END_IF

IF PWM_Y2_SET<TO_INT(PAR_Y1_1_NegFull )THEN
	PWM_Y2_SET:=TO_INT(PAR_Y1_1_NegFull);
END_IF

IF(PWM_Y1_SET>1000) THEN
	PWM_Y1_SET := 300;
END_IF

IF(PWM_Y2_SET>1000) THEN
	PWM_Y2_SET := 300;
END_IF
(*电控马达动力头变量控制*)
(*
DonglitouPressureSub:=UINT_TO_INT(CANO_DonglitouPressure - CANO_DonglitouPressure_last);
//只需小范围波动滤波
	IF(DonglitouPressureSub>10 OR DonglitouPressureSub<-10)THEN 
		DonglitouPressure_ChangeBool:=TRUE;
	ELSE
		DonglitouPressure_ChangeBool:=FALSE;
	END_IF

	TIME_LvBo3(IN:=DonglitouPressure_ChangeBool,PT:=T#500MS);
	IF(TIME_LvBo3.Q )THEN
		CANO_DonglitouPressure_last:=CANO_DonglitouPressure;
	END_IF	
IF(PWM_JOYX_R_UP>10 OR PWM_JOYX_R_DOWN>10)THEN
	IF(CANO_DonglitouPressure_last>260) THEN
	PWM_Y34_SET_Target :=380;   
	ELSIF(CANO_DonglitouPressure_last>240) THEN   
	PWM_Y34_SET_Target :=508;  
	ELSIF(CANO_DonglitouPressure_last>220) THEN   
	PWM_Y34_SET_Target :=605;  
	ELSIF(CANO_DonglitouPressure_last>200) THEN   
	PWM_Y34_SET_Target :=703;  
	ELSIF(CANO_DonglitouPressure_last>180) THEN   
	PWM_Y34_SET_Target :=801;  
	ELSIF(CANO_DonglitouPressure_last>160) THEN   
	PWM_Y34_SET_Target :=899;  
	ELSE
	PWM_Y34_SET_Target :=1100;  
	END_IF
ELSE
	PWM_Y34_SET_Target :=1100;  
END_IF

IF(CANO_DonglitouPressure<20) THEN
	JianGE22:=10;
ELSE
	JianGE22:=1.5;
END_IF
IF PWM_Y34_SET>PWM_Y34_SET_Target THEN
	PWM_Y34_SET := REAL_TO_UINT(UINT_TO_REAL(PWM_Y34_SET)-JianGE22);
END_IF

IF(PWM_Y34_SET<=PWM_Y34_SET_Target) THEN
	PWM_Y34_SET:=REAL_TO_UINT(UINT_TO_REAL(PWM_Y34_SET)+JianGE22);
END_IF


//H.M.L档
IF(CANI_DonglitouMSwitch) THEN
	IF(CANO_DonglitouPressure>280) THEN
		PWM_Y34_SET_Target :=380;  
	ELSIF(CANO_DonglitouPressure>270) THEN   
		PWM_Y34_SET_Target :=459;  
	ELSIF(CANO_DonglitouPressure>260) THEN   
		PWM_Y34_SET_Target :=508;  
	ELSIF(CANO_DonglitouPressure>250) THEN   
		PWM_Y34_SET_Target :=557;  
	ELSIF(CANO_DonglitouPressure>240) THEN   
		PWM_Y34_SET_Target :=605;  
	ELSIF(CANO_DonglitouPressure>230) THEN   
		PWM_Y34_SET_Target :=654;  
	ELSE
		PWM_Y34_SET_Target:=703;
	END_IF
END_IF

IF(CANI_DonglitouHSwitch) THEN
	PWM_Y34_SET_Target := 200;
END_IF

IF(DIH_SA15)THEN
	IF(PWM_Y34_SET_Target<600)THEN
		PWM_Y34_SET_Target:=600;
	END_IF
END_IF

IF PWM_Y34_SET>=PWM_Y34_SET_Target THEN
	PWM_Y34_SET := PWM_Y34_SET_Target;
END_IF

IF DIL_SQ3 THEN
	PWM_Y34_SET:=200;
END_IF

IF(PWM_Y34_SET>2000) THEN
	PWM_Y34_SET := 2000;
END_IF
*)
//液控马达
//动力头调速
Rtrig_d1(CLK:=CANI_DonglitouADDSwitch);
Rtrig_d2(CLK:=CANI_DonglitouSUBSwitch);
IF (Rtrig_d1.Q AND DI_LHandle_SB1 )THEN
	IF(CANI_DonglitouHSwitch AND NOT CANI_DonglitouLSwitch AND NOT CANI_DonglitouMSwitch)THEN
		PAR_MotorChioce_H_PWM:=PAR_MotorChioce_H_PWM+10;
	ELSIF(CANI_DonglitouMSwitch AND NOT CANI_DonglitouLSwitch AND NOT CANI_DonglitouHSwitch)THEN
		PAR_MotorChioce_M_PWM:=PAR_MotorChioce_M_PWM+10;
	ELSE
		PAR_MotorChioce_L_PWM:=PAR_MotorChioce_L_PWM+10;
	END_IF
ELSIF(Rtrig_d2.Q AND DI_LHandle_SB1)THEN
	IF(CANI_DonglitouHSwitch AND NOT CANI_DonglitouLSwitch AND NOT CANI_DonglitouMSwitch)THEN
		IF PAR_MotorChioce_H_PWM<20 THEN
			PAR_MotorChioce_H_PWM:=20;
		END_IF
		PAR_MotorChioce_H_PWM:=PAR_MotorChioce_H_PWM-10;
	ELSIF(CANI_DonglitouMSwitch AND NOT CANI_DonglitouLSwitch AND NOT CANI_DonglitouHSwitch)THEN
		IF PAR_MotorChioce_M_PWM<20 THEN
			PAR_MotorChioce_M_PWM:=20;
		END_IF
		PAR_MotorChioce_M_PWM:=PAR_MotorChioce_M_PWM-10;
	ELSE

		IF PAR_MotorChioce_L_PWM<20 THEN
			PAR_MotorChioce_L_PWM:=20;
		END_IF
		PAR_MotorChioce_L_PWM:=PAR_MotorChioce_L_PWM-10;
	END_IF
END_IF

	IF(CANI_DonglitouHSwitch AND NOT CANI_DonglitouLSwitch AND NOT CANI_DonglitouMSwitch)THEN
		PWM_Y34_SET:=PAR_MotorChioce_H_PWM;
	ELSIF(CANI_DonglitouMSwitch AND NOT CANI_DonglitouLSwitch AND NOT CANI_DonglitouHSwitch)THEN
		PWM_Y34_SET:=PAR_MotorChioce_M_PWM;
	ELSE
		PWM_Y34_SET:=PAR_MotorChioce_L_PWM;
	END_IF

PressLvBo_TON(IN:=CANO_ZhuJuanPressure>310,PT:=T#300MS);
PressLvBo_TON1(IN:=CANO_ZhuJuanPressure>290 AND CANO_ZhuJuanPressure<=310,PT:=T#300MS);
PressLvBo_TON2(IN:=CANO_ZhuJuanPressure>270 AND CANO_ZhuJuanPressure<=290,PT:=T#300MS);
PressLvBo_TON3(IN:=CANO_ZhuJuanPressure>250 AND CANO_ZhuJuanPressure<=270,PT:=T#300MS);
IF(CANO_ZhuJuanPressure>310 AND PressLvBo_TON.Q) OR P31_Flag THEN
        PWM_Y33_SET_Target :=230;   //排量200
        P31_Flag:=TRUE;
        IF (CANO_ZhuJuanPressure<270) THEN
                P31_Flag:=FALSE;        
        END_IF
ELSIF(CANO_ZhuJuanPressure>290 AND PressLvBo_TON1.Q) OR P29_Flag THEN   
        PWM_Y33_SET_Target :=267;   //排量180
        P29_Flag:=TRUE; 
        IF (CANO_ZhuJuanPressure<250) THEN
                P29_Flag:=FALSE; 
        END_IF
ELSIF(CANO_ZhuJuanPressure>270 AND PressLvBo_TON2.Q) OR P27_Flag THEN   
        PWM_Y33_SET_Target :=304;  //排量160
        P27_Flag:=TRUE;
        IF (CANO_ZhuJuanPressure<230) THEN
                P27_Flag:=FALSE; 
        END_IF
ELSIF(CANO_ZhuJuanPressure>250 AND PressLvBo_TON3.Q) OR P25_Flag THEN //压力小于270   
        PWM_Y33_SET_Target :=340;  //排量140
        P25_Flag:=TRUE; 
        IF (CANO_ZhuJuanPressure<210) THEN
                P25_Flag:=FALSE; 
        END_IF
ELSE //(CANO_ZhuJuanPressure<=250) THEN
        PWM_Y33_SET_Target :=370;
END_IF

IF NOT MainWinch_move THEN
    P25_Flag:=FALSE;
    P27_Flag:=FALSE;
    P29_Flag:=FALSE; 
    P31_Flag:=FALSE;        
END_IF       


IF BiaoZHI_MainWinchUp THEN  //单主卷下放370马达电流
 	PWM_Y33_SET_Target:=370;
END_IF

IF PWM_Y33_SET>=PWM_Y33_SET_Target THEN
	PWM_Y33_SET := PWM_Y33_SET_Target;
END_IF
	
IF(PWM_Y33_SET<PWM_Y33_SET_Target) THEN
	PWM_Y33_SET:=REAL_TO_UINT(UINT_TO_REAL(PWM_Y33_SET)+JianGE6);
END_IF

IF DIL_SQ3 THEN
	PWM_Y33_SET:=0;
END_IF
//动力头抛土
(******************抛土控制******************)
(*自动抛土*)
	IF DI_RHandle_SB6 AND PowerHead_move THEN
		IF CANO_JiayaPressure>80 OR Rotation_move THEN     //抛土模式做了延时，防止3泵工作熄火
			PWM_Y1_SET:=450;//此值要确认抛土效果 
			PWM_Y2_SET:=450;
		ELSE
			PWM_Y1_SET:=UINT_TO_INT(PAR_ValveC_PosFull);
			PWM_Y2_SET:=UINT_TO_INT(PAR_ValveC_PosFull);
		END_IF
		PWM_Y39_SET:=1300;
		PWM_Y40_SET:=1300;
		DonglitouBlink(ENABLE:=TRUE,TIMELOW:=T#300MS,TIMEHIGH:=T#300MS);
		IF DonglitouBlink.OUT THEN
			PWM_Y12_SET:=PAR_Valve1_PosFull;
			PWM_Y14_SET:=PAR_Valve2_PosFull;
			PWM_Y61_SET:=PAR_Valve1_PosFull;
			PWM_Y11_SET:=0;
			PWM_Y13_SET:=0;
			PWM_Y60_SET:=0;
		ELSE
			DonglitouBlink_biaozhi:=FALSE;
			PWM_Y12_SET:=0;
			PWM_Y14_SET:=0;
			PWM_Y61_SET:=0;
			PWM_Y11_SET:=PAR_Valve1_PosFull;
			PWM_Y13_SET:=PAR_Valve2_PosFull;
			PWM_Y60_SET:=PAR_Valve1_PosFull;
		END_IF
	END_IF
	
	
	(*主卷自动抖土*)
	(*IF DI_LHandle_SB2 AND PowerHead_move THEN
		PWM_Y1_SET:=TO_INT(PAR_ValveD_PosFull);
		PWM_Y2_SET:=TO_INT(PAR_ValveD_PosFull);
		PWM_Y39_SET:=1200;
		PWM_Y40_SET:=1200;
		DonglitouBlink(ENABLE:=TRUE,TIMELOW:=T#400MS,TIMEHIGH:=T#400MS);
		IF DonglitouBlink.OUT THEN
			PWM_Y7_SET:=PAR_Valve1_PosFull;
			PWM_Y9_SET:=PAR_Valve2_PosFull;
		ELSE
			PWM_Y7_SET:=0;
			PWM_Y9_SET:=0;
		END_IF
	END_IF*)



(*冷却风扇控制*)
IF NOT CANI_ColdFunSwitch  THEN
	IF(CANO_Hyd_Tem>60)THEN
		PWM_Y49_SET := PAR_ValveD_NegFull;
	END_IF
	
	IF(CANO_Hyd_Tem<60)THEN
		PWM_Y49_SET := 0;		
	END_IF
ELSE
	PWM_Y49_SET := PAR_ValveD_NegFull;
END_IF

(*主卷浮动*)
IF((DIH_SA8 OR DI_LHandle_SB3 OR CANI_Button_FloatSwitch) AND CANI_MaiWinFloatSwitch AND (NOT DIL_SQ3)) THEN
	DOH_Y55:=TRUE;
	DOH_Y56:=TRUE;
ELSE
	DOH_Y55:=FALSE;
	DOH_Y56:=FALSE;
END_IF

(*主卷开锁*)
(*IF MainWinch_move AND (NOT PowerHead_move )AND (PWM_JOYY_L_UP<500 AND PWM_JOYY_L_DOWN=0) AND CANO_ZhuJuanPressure<100 THEN
	DOH_Y56:=TRUE;
END_IF*)

IF(UIGroupVoltage0<2000 OR UIGroupVoltage1<2000 OR UIGroupVoltage2<2000 
   OR UIGroupVoltage3<2000 OR UIGroupVoltage4<2000 OR UIGroupVoltage5<2000) THEN
	reset111:=TRUE;
ELSE
	reset111:=FALSE;
END_IF
(*
IF Paotu_Modle THEN
	PWM_Y1_SET:=UINT_TO_INT(testpaotu);//PAR_ValveC_PosFull
	PWM_Y2_SET:=UINT_TO_INT(testpaotu);
END_IF
*)

IF Paotu_Modle THEN
	IF CANO_JiayaPressure>80 OR Rotation_move THEN     //抛土模式做了延时，防止3泵工作熄火
		PWM_Y1_SET:=450;//此值要确认抛土效果 
		PWM_Y2_SET:=450;
	ELSE
		PWM_Y1_SET:=UINT_TO_INT(PAR_ValveC_PosFull);
		PWM_Y2_SET:=UINT_TO_INT(PAR_ValveC_PosFull);
	END_IF
	PWM_Y39_SET:=1300;
	PWM_Y40_SET:=1300;
END_IF

END_PROGRAM

// StandardPLC/Application/MOVE/MastControl
PROGRAM MastControl
VAR
	VarCurrentMax	:INT;
	VarCurrentMin	:INT;
	VarU16		 	:UINT;
	VarTempInt32 	:int;
	VarFloat32A: REAL;
	VarFloat32B: REAL;
	i: UINT;
	LibSqrt_input: REAL;
	VarMastAutoOk: BOOL;
	VarMastAutoStep: UINT;
	VarTempInt16: INT;
	VarMastTempLoopCount :UINT;
	VarMastAutoOk_1: BOOL;
	MastAutoTime:TON;
	VarAutoTiaoPingTiaoJian: BOOL;
	Joyy_Error: BOOL;
	Joyx_Error: BOOL;
	Error_x:TON;
	Error_y:TON;
	angle_xy:censor_cali;
	VarJoyX100_1:UINT;
	VarJoyY100_1:UINT;
	VarFloat32A1:REAL;
	Mast_BuCang:INT;
	VarMastA_target: INT;
	VarMastA_1: INT;
	ftp_2s_1:TON;
	ftp_2s_2:TON;
END_VAR

(*手柄输入*)
IF(NOT CANI_WorkModeSwitch) THEN (*调整档*)
	VarTempInt32:=UINT_TO_INT(AI_JOYY)-2500;
	IF(VarTempInt32>2500) THEN
		VarTempInt32 := 2500;
	ELSIF(VarTempInt32<-2500) THEN
		VarTempInt32 := -2500;
	ELSIF(VarTempInt32>-150 AND VarTempInt32<150) THEN
		VarTempInt32 := 0;
	END_IF
 		VarJoyY:=VarTempInt32; //-2500～+2500
ELSE
	VarJoyY:=0;
END_IF

IF(NOT CANI_WorkModeSwitch) THEN (*调整档*)
	VarTempInt32:=UINT_TO_INT(AI_JOYX)-2500;
	IF(VarTempInt32>2500) THEN
		VarTempInt32 := 2500;
	ELSIF(VarTempInt32<-2500) THEN
		VarTempInt32 := -2500;
	ELSIF(VarTempInt32>-150 AND VarTempInt32<150) THEN
		VarTempInt32 := 0;
	END_IF
 		VarJoyX:=VarTempInt32; //-2500～+2500
ELSE
	VarJoyX:=0;
END_IF

(*手柄故障报警*)
IF(AI_JOYY<2 OR AI_JOYY>4980)THEN
	Joyy_Error:=TRUE;
ELSE
	Joyy_Error:=FALSE;
END_IF

IF(AI_JOYX<2 OR AI_JOYX>4980)THEN
	Joyx_Error:=TRUE;
ELSE
	Joyx_Error:=FALSE;
END_IF
Error_x(IN:=Joyx_Error,PT:=T#600S);
Error_y(IN:=Joyy_Error,PT:=T#600S);
IF(Error_x.Q OR Error_y.Q)THEN
	CANO_SensorError_Joy:=TRUE;
ELSE
	CANO_SensorError_Joy:=FALSE;
END_IF

(*PWM_OUTPUT*)
	VarMastA_ := VarMastA;//-100 ~ +100
	VarMastB_ := VarMastB;//-100 ~ +100
	
	IF (VarMastA_ > 0) THEN
		VarCurrentMax := UINT_TO_INT(PAR_Y27_PosFull);
		VarCurrentMin := UINT_TO_INT(PAR_Y27_NegFull);
		VarMastA_ := VarMastA_*(VarCurrentMax - VarCurrentMin)/100 + VarCurrentMin;
	
	ELSIF(VarMastA_ < 0) THEN
		VarCurrentMax := UINT_TO_INT(PAR_Y28_PosFull);
		VarCurrentMin := UINT_TO_INT(PAR_Y28_NegFull);
		VarMastA_ := VarMastA_*(VarCurrentMax - VarCurrentMin)/100 - VarCurrentMin;
	END_IF
	
	IF (VarMastB_ > 0) THEN
		VarCurrentMax := UINT_TO_INT(PAR_Y29_PosFull);
		VarCurrentMin := UINT_TO_INT(PAR_Y29_NegFull);
		VarMastB_ := VarMastB_*(VarCurrentMax - VarCurrentMin)/100 + VarCurrentMin;
	
	ELSIF(VarMastB_ < 0) THEN
		VarCurrentMax := UINT_TO_INT(PAR_Y30_PosFull);
		VarCurrentMin := UINT_TO_INT(PAR_Y30_NegFull);
		VarMastB_ := VarMastB_*(VarCurrentMax - VarCurrentMin)/100 - VarCurrentMin;
	END_IF

	IF(VarMastA_>=0) THEN  //伸
		VarU16 := INT_TO_UINT(VarMastA_);  //VarCurrentMin～VarCurrentMax
		IF (VarMastWorkMode=3) THEN
			IF(PWM_Y27_SET<VarU16) THEN
				PWM_Y27_SET := PWM_Y27_SET + 1;
				IF(PWM_Y27_SET<400) THEN
					PWM_Y27_SET := PWM_Y27_SET + 10;
				END_IF				
			ELSIF(PWM_Y27_SET>VarU16)THEN
				PWM_Y27_SET:=PWM_Y27_SET-1;
			END_IF
		ELSE
			PWM_Y27_SET := VarU16;
		END_IF
		PWM_Y28_SET := 0;
	ELSE
		PWM_Y27_SET := 0;
	    VarU16 := INT_TO_UINT(-VarMastA_);
	    IF(VarMastWorkMode=3)  THEN
			IF(PWM_Y28_SET<VarU16) THEN
				PWM_Y28_SET := PWM_Y28_SET + 1;
		    	IF(PWM_Y28_SET<400) THEN
		    		PWM_Y28_SET:=PWM_Y28_SET + 10;
		    	END_IF
		    ELSIF(PWM_Y28_SET>VarU16) THEN
		    	PWM_Y28_SET:=PWM_Y28_SET-1;
			END_IF
		ELSE
			PWM_Y28_SET := VarU16;
		END_IF
	END_IF
		
	IF(VarMastB_>=0) THEN  //伸
		VarU16 := INT_TO_UINT(VarMastB_);  //VarCurrentMin～VarCurrentMax
		IF (VarMastWorkMode=3) THEN
			IF(PWM_Y29_SET<VarU16) THEN
				PWM_Y29_SET := PWM_Y29_SET + 1;
				IF(PWM_Y29_SET<400) THEN
					PWM_Y29_SET := PWM_Y29_SET + 10;
				END_IF				
			ELSIF(PWM_Y29_SET>VarU16)THEN
				PWM_Y29_SET:=PWM_Y29_SET-1;
			END_IF
		ELSE
			PWM_Y29_SET := VarU16;
		END_IF
		PWM_Y30_SET := 0;
	ELSE
		PWM_Y29_SET := 0;
	    VarU16 := INT_TO_UINT(-VarMastB_);
	    IF(VarMastWorkMode=3)  THEN
			IF(PWM_Y30_SET<VarU16) THEN
				PWM_Y30_SET := PWM_Y30_SET + 1;
		    	IF(PWM_Y30_SET<400) THEN
		    		PWM_Y30_SET:=PWM_Y30_SET + 10;
		    	END_IF
		    ELSIF(PWM_Y30_SET>VarU16) THEN
		    	PWM_Y30_SET:=PWM_Y30_SET-1;
			END_IF
		ELSE
			PWM_Y30_SET := VarU16;
		END_IF
	END_IF

(*计算手柄的角度和长度*)
	VarJoyX100:=VarJoyX*100/2500;//-100~100
	VarJoyY100:=VarJoyY*100/2500;//-100~100
	VarGama := 90;
	
	VarJoyX100_1:=INT_TO_UINT(ABS(VarJoyX100)+1);
	VarJoyY100_1:=INT_TO_UINT(ABS(VarJoyY100)+1);
	VarFloat32A1 := UINT_TO_REAL(VarJoyY100_1)/UINT_TO_REAL(VarJoyX100_1);

	VarGama:=REAL_TO_UINT((ATAN(VarFloat32A1))*180/3.14);
	(*IF(VarJoyX<>0) THEN
		VarFloat32A := VarJoyX;
		VarFloat32B := VarJoyY;
		VarFloat32A := VarFloat32B/VarFloat32A;
		IF (VarFloat32A < 0 ) THEN
			VarFloat32A:= -VarFloat32A;
		END_IF

		FOR i:=0 TO 90 DO
			IF(VarFloat32A  <= TAN(i)) THEN
				VarGama := i;
			END_IF
		END_FOR
	END_IF*)
	
	VarFloat32A := VarJoyX100;
	VarFloat32B := VarJoyY100;

	LibSqrt_input:= VarFloat32A*VarFloat32A + VarFloat32B*VarFloat32B;
	VarLengthC:=SQRT(LibSqrt_input);
	IF(VarLengthC>100)THEN VarLengthC:=100; END_IF
	
	//转换
	VarAngleXDelta :=  (UINT_TO_INT(CANO_ANGLE_X)-9000) ;//转换-90°-90° 
	VarAngleYDelta :=  (UINT_TO_INT(CANO_ANGLE_Y)-9000) ;//转换-90°-90°
	
	IF(VarAngleXDelta>20 AND VarAngleXDelta<=30) OR (VarAngleXDelta<-20 AND VarAngleXDelta>=-30)THEN
		Mast_BuCang := 2;
	ELSIF(VarAngleXDelta>30 AND VarAngleXDelta<=40) OR (VarAngleXDelta<-30 AND VarAngleXDelta>=-40)THEN
		Mast_BuCang := 4;
	ELSIF(VarAngleXDelta>40 AND VarAngleXDelta<=50) OR (VarAngleXDelta<-40 AND VarAngleXDelta>=-50)THEN
		Mast_BuCang := 6;
	ELSIF(VarAngleXDelta>50 AND VarAngleXDelta<=60) OR (VarAngleXDelta<-50 AND VarAngleXDelta>=-60)THEN
		Mast_BuCang := 8;
	ELSIF(VarAngleXDelta>60 AND VarAngleXDelta<=70) OR (VarAngleXDelta<-60 AND VarAngleXDelta>=-70)THEN
		Mast_BuCang := 10;
	ELSIF(VarAngleXDelta>70 AND VarAngleXDelta<=80) OR (VarAngleXDelta<-70 AND VarAngleXDelta>=-80)THEN
		Mast_BuCang := 12;
	ELSIF(VarAngleXDelta>80 AND VarAngleXDelta<=90) OR (VarAngleXDelta<-80 AND VarAngleXDelta>=-90)THEN
		Mast_BuCang := 14;
	ELSIF(VarAngleXDelta>90 ) OR (VarAngleXDelta<-90 )THEN
		Mast_BuCang := 15;
	END_IF
	
	IF(VarAngleYDelta<-6000) THEN
		Mast_BuCang:=0;
	END_IF
	ftp_2s_1(IN:=(VarAngleXDelta>20),PT:=T#2S);
	ftp_2s_2(IN:=(VarAngleXDelta<-20),PT:=T#2S);
	//计算油缸电流输出值
	IF((NOT DIL_SQ3) AND (NOT CANI_WorkModeSwitch) AND (NOT VarGpsSystemLockedState)) THEN
		//限位模式
		IF(VarMastWorkMode=1) THEN
			IF(DIH_JOY) THEN
				IF((NOT DIH_SQ5) AND (NOT DIH_SQ6))  THEN//限位传感器错误
					VarMastA := 0;
					VarMastB := 0;
				ELSIF( (((NOT DIH_SQ5) OR TooLowX_angle)AND(VarJoyX100>0)) OR  //右限位报警或者X倾角小于4度
				         (((NOT DIH_SQ6) OR TooHighX_angle)AND(VarJoyX100<0))) THEN
					VarMastA := VarJoyX100;
					VarMastB := -VarMastA;
				ELSIF(TooHighY AND VarJoyY100<0) THEN
					VarMastA := VarJoyY;
					VarMastB := VarMastA;
				ELSE
					VarMastA := 0;
					VarMastB := 0;
				END_IF
			ELSE
				VarMastA := 0;
				VarMastB := 0;
			END_IF
			VarMastA_target:=0;
			VarMastA_1:=VarMastA*12;
		//手动模式	
		ELSIF (VarMastWorkMode=2) THEN
			IF (DIH_JOY) THEN
				//死区
				IF((VarJoyX100>=-5 AND VarJoyX100<=5)AND(VarJoyY100>=-5 AND VarJoyY100<=5)) THEN
					VarMastA := 0;
					VarMastB := 0;
				//沿Y轴
			//沿Y轴
				ELSIF((VarJoyX100>-45 AND VarJoyX100<45)AND(VarJoyY100<-5 OR VarJoyY100>5)) THEN
					VarMastA := VarJoyY100;
					VarMastB := VarMastA;
					
					IF(VarJoyY100>5)THEN
						IF(ftp_2s_1.Q) THEN
							IF(VarJoyY100>Mast_BuCang) THEN
								VarMastA:=VarJoyY100 - Mast_BuCang;
							END_IF
							VarMastB := VarJoyY100 + Mast_BuCang;
						ELSIF (ftp_2s_2.Q) THEN
							IF(VarJoyY100>Mast_BuCang) THEN
								VarMastB:=VarJoyY100 - Mast_BuCang;
							END_IF
							VarMastA := VarJoyY100 + Mast_BuCang;
						END_IF
					ELSIF (VarJoyY100<-5)THEN
						IF(ftp_2s_1.Q) THEN
							VarMastA:=VarJoyY100 - Mast_BuCang;
							IF(VarJoyY100 + Mast_BuCang)<0 THEN
								VarMastB:= VarJoyY100 + Mast_BuCang;
							END_IF
						ELSIF (ftp_2s_2.Q) THEN
							VarMastB:=VarJoyY100 - Mast_BuCang;
							IF(VarJoyY100 + Mast_BuCang)<0 THEN
								VarMastA := VarJoyY100 + Mast_BuCang;
							END_IF
						END_IF
					END_IF

				//沿X轴
				ELSIF((VarJoyY100>-15 AND VarJoyY100<15)AND(VarJoyX100<-5 OR VarJoyX100>5)) THEN
					
					IF (VarJoyX100>30) THEN
						VarJoyX100:=30;
					END_IF
					IF (VarJoyX100<-30) THEN
						VarJoyX100:=-30;
					END_IF
					
					VarMastA_target := VarJoyX100*10;
					IF(VarMastA_target>4 AND VarMastA_1<=VarMastA_target) THEN
						VarMastA_1 := VarMastA_1 + 3;
					ELSIF (VarMastA_target>4 AND VarMastA_1>VarMastA_target) THEN
						VarMastA_1 :=VarMastA_1 - 3; 
					END_IF
					IF(VarMastA_target<-4 AND VarMastA_1>=VarMastA_target) THEN
						VarMastA_1 := VarMastA_1 - 3;
					ELSIF(VarMastA_target<-4 AND VarMastA_1<VarMastA_target) THEN
						VarMastA_1 := VarMastA_1 + 3;
					END_IF
					VarMastA := VarMastA_1/10;
					VarMastB := -VarMastA;
				(*ELSE
					//手柄动作的角度小于23度,桅杆总的趋势是AB值相反
					IF (VarGama<23.0) THEN
						//X动作大于Y动作,并且XY都为正,第一象限,A油缸伸,B油缸缩,但A比B大,应使角度朝右前运动
						IF(VarJoyX100>0 AND VarJoyY100>0) THEN
							VarMastA := REAL_TO_INT(VarLengthC*(VarGama+23.0)/46.0);
							VarMastB := REAL_TO_INT(VarLengthC*(VarGama-23.0)/46.0);
						//X动作大于Y动作,并且X为正,Y为负,第四象限,A油缸伸,B油缸缩,但A比B小,应使角度朝右后运动
						ELSIF(VarJoyX100>0 AND VarJoyY100<0) THEN
							VarMastA := REAL_TO_INT(VarLengthC*(+23.0-VarGama)/46.0);
							VarMastB := REAL_TO_INT(VarLengthC*(-23.0-VarGama)/46.0);
						//X动作大于Y动作,并且X为负,Y为正,第二象限,A油缸缩,B油缸伸,但A比B小,应使角度朝左前运动
						ELSIF(VarJoyX100<0 AND VarJoyY100>0) THEN
							VarMastA := REAL_TO_INT(VarLengthC*(VarGama-23.0)/46.0);
							VarMastB := REAL_TO_INT(VarLengthC*(VarGama+23.0)/46.0);
						//X动作大于Y动作,并且X为负,Y为负,第三象限,A油缸缩,B油缸伸,但A比B大,应使角度朝左后运动
						ELSIF(VarJoyX100<0 AND VarJoyY100<0) THEN
							VarMastA := REAL_TO_INT(VarLengthC*(-23.0-VarGama)/46.0);
							VarMastB := REAL_TO_INT(VarLengthC*(+23.0-VarGama)/46.0);
						//异常
						ELSE
							VarMastA := 0;
							VarMastB := 0;
						END_IF
					//手柄动作的角度大于23度,桅杆总得趋势是AB值相同
					ELSE
						//XY都为正,第一象限,A伸,B伸,但A比B大,应使角度朝前右运动
						IF(VarJoyX100>0 AND VarJoyY100>0) THEN
							VarMastA := REAL_TO_INT(VarLengthC*(180.0-VarGama-23.0)/134.0);
							VarMastB := REAL_TO_INT(VarLengthC*(VarGama-23.0)/134.0);
						//X为负,Y为正,第二象限,A伸,B伸,但A比B小,应使角度朝前左运动
						ELSIF(VarJoyX100<0 AND VarJoyY100>0) THEN
							VarMastA := REAL_TO_INT(VarLengthC*(VarGama-23.0)/134.0);
							VarMastB := REAL_TO_INT(VarLengthC*(180.0-VarGama-23.0)/134.0);
						//X为负,Y为负,第三象限,A缩,B缩,但A比B大,应使角度朝后左运动
						ELSIF(VarJoyX100<0 AND VarJoyY100<0) THEN
							VarMastA := REAL_TO_INT(VarLengthC*(-180.0+VarGama+23.0)/134.0);
							VarMastB := REAL_TO_INT(VarLengthC*(23.0-VarGama)/134.0);
						//X为正,Y为负,第四象限,A缩,B缩,但A比B小,应使角度朝后后运动
						ELSIF(VarJoyX100>0 AND VarJoyY100<0) THEN
							VarMastA := REAL_TO_INT(VarLengthC*(23.0-VarGama)/134.0);
							VarMastB := REAL_TO_INT(VarLengthC*(-180.0+VarGama+23.0)/134.0);
						//异常
						ELSE
							VarMastA := 0;
							VarMastB := 0;
						END_IF
					END_IF*)
				END_IF
			//未按下手柄
			else
				VarMastA := 0;
				VarMastB := 0;
				VarMastA_target :=0;
				VarMastA_1:=0;
			END_IF
			
			//显示屏控制  X+/X-/Y+/Y-
			IF(CANI_Button_LEVER_XPlus)THEN
				VarMastA := 25;
				VarMastB := -18;
			ELSIF(CANI_Button_LEVER_XSubtract)THEN
				VarMastA := -25;
				VarMastB := 18;
			ELSIF(CANI_Button_LEVER_YPlus) THEN
				VarMastA := 30;
				VarMastB := 30;
			ELSIF(CANI_Button_LEVER_YSubtract) THEN
				VarMastA := -30;
				VarMastB := -30;
			END_IF	
	
			//显示屏控制  左伸/左缩/右伸/右缩
			IF(CANI_Button_Debug_LStretchOut) THEN
				VarMastA := 30;
				VarMastB := 0;	
			ELSIF(CANI_Button_Debug_LRetraction) THEN
				VarMastA :=-30;
				VarMastB := 0;	
			ELSIF(CANI_Button_Debug_RStretchOut) THEN
				VarMastA :=0;
				VarMastB := 30;	
			ELSIF(CANI_Button_Debug_RRetraction) THEN
				VarMastA :=0;
				VarMastB :=-30;	
			END_IF
		//自动模式
		ELSIF(VarMastWorkMode=3) THEN
			//已经调平
			IF(VarMastAutoOk)THEN
				VarMastA := 0;
				VarMastB := 0;
			ELSE
				CASE VarMastAutoStep OF
				0,2,4,6,8:
					IF(VarMastA>=2) THEN
						VarMastA := VarMastA - 2;
					ELSIF(VarMastA<=-2) THEN
						VarMastA := VarMastA + 2;
					ELSE
						VarMastA := 0;
					END_IF
					
					IF(VarMastB>=2) THEN
						VarMastB := VarMastB - 2;
					ELSIF(VarMastB<=-2) THEN
						VarMastB := VarMastB + 2;
					ELSE 
						VarMastB := 0;
					END_IF
				
					IF(VarMastA=0 AND VarMastB=0) THEN
						VarMastAutoStep:=VarMastAutoStep + 1;
					END_IF
				//将X大于零方向回归;A-,B+
				1:
					IF(VarAngleXDelta>10) THEN  //每单位0.01度
						VarTempInt16:= VarAngleXDelta/30*8 + 5;
						IF(VarTempInt16>40) THEN
							VarTempInt16:=40;
						END_IF
						//20131105*add****************start
						IF(VarMastTempLoopCount>10)THEN    //取10次循环
							IF(VarMastA>-VarTempInt16) THEN
								VarMastA :=VarMastA - 1;
							ELSE
								VarMastA := -VarTempInt16;
							END_IF
							VarMastTempLoopCount:=0;
						END_IF
						VarMastTempLoopCount:=VarMastTempLoopCount + 1;
						//*****************************end
						VarMastB := -VarMastA;//B+  //20140225...修改
					ELSE
							VarMastAutoStep:=VarMastAutoStep + 1;
					END_IF
				//将X小于零方向归零;A+,B-
				3:
					IF(VarAngleXDelta<-10) THEN  //每单位0.01度
						VarTempInt16:= VarAngleXDelta/30*8 - 5;
						IF(VarTempInt16<-40) THEN
							VarTempInt16:=-40;
						END_IF
						//20131105*add****************start
						IF(VarMastTempLoopCount>10)THEN    //取10次循环
							IF(VarMastA<-VarTempInt16) THEN
								VarMastA :=VarMastA + 1;
							ELSE
								VarMastA := -VarTempInt16;
							END_IF
							VarMastTempLoopCount:=0;
						END_IF
						VarMastTempLoopCount:=VarMastTempLoopCount + 1;
						//*****************************end
						VarMastB := -VarMastA;//B+  //20140225...修改
					ELSE
							VarMastAutoStep:=VarMastAutoStep + 1;
					END_IF
				//将Y大于零方向归零;A-,B-
				5:
					IF(VarAngleYDelta>10) THEN  //每单位0.01度
						VarTempInt16:= VarAngleYDelta/30*8 + 5;
						IF(VarTempInt16>40) THEN
							VarTempInt16:=40;
						END_IF
						//20131105*add****************start
						IF(VarMastTempLoopCount>10)THEN    //取10次循环
							IF(VarMastA>-VarTempInt16) THEN
								VarMastA :=VarMastA - 1;
							ELSE
								VarMastA := -VarTempInt16;
							END_IF
							VarMastTempLoopCount:=0;
						END_IF
						VarMastTempLoopCount:=VarMastTempLoopCount + 1;
						//*****************************end
						VarMastB := VarMastA;//B+  //20140225...修改
					ELSE
							VarMastAutoStep:=VarMastAutoStep + 1;
					END_IF
				//将Y小于零方向归零;A+,B+
				7:
					IF(VarAngleYDelta<-10) THEN  //每单位0.01度
						VarTempInt16:= VarAngleYDelta/30*8 - 10;
						IF(VarTempInt16<-40) THEN
							VarTempInt16:=-40;
						END_IF
						//20131105*add****************start
						IF(VarMastTempLoopCount>10)THEN    //取10次循环
							IF(VarMastA<-VarTempInt16) THEN
								VarMastA :=VarMastA + 1;
							ELSE
								VarMastA := -VarTempInt16;
							END_IF
							VarMastTempLoopCount:=0;
						END_IF
						VarMastTempLoopCount:=VarMastTempLoopCount + 1;
						//*****************************end
						VarMastB := VarMastA;//B+  //20140225...修改
					ELSE
						VarMastAutoStep:=VarMastAutoStep + 1;
					END_IF 
					//微调
				9:
					IF(VarAngleXDelta>10) THEN
						IF(VarAngleXDelta>30)THEN
							VarTempInt16:=16;
						ELSE
							VarTempInt16:=8;
						END_IF
						IF(VarMastTempLoopCount>10)THEN    //取10次循环
							IF(VarMastA>-VarTempInt16) THEN
								VarMastA :=VarMastA - 1;
							ELSE
								VarMastA := -VarTempInt16;
							END_IF
							VarMastTempLoopCount:=0;
						END_IF
						VarMastTempLoopCount:=VarMastTempLoopCount + 1;
						VarMastB := -VarMastA;
					ELSIF(VarAngleXDelta<-10)THEN
						IF(VarAngleXDelta<-30)THEN
							VarTempInt16:=16;
						ELSE
							VarTempInt16:=8;
						END_IF
						IF(VarMastTempLoopCount>10)THEN    //取10次循环
							IF(VarMastA<-VarTempInt16) THEN
								VarMastA :=VarMastA + 1;
							ELSE
								VarMastA := VarTempInt16;
							END_IF
							VarMastTempLoopCount:=0;
						END_IF
						VarMastTempLoopCount:=VarMastTempLoopCount + 1;
						VarMastB := -VarMastA;
					ELSIF(VarAngleYDelta>10)THEN
						IF(VarAngleYDelta>30)THEN
							VarTempInt16:=16;
						ELSE
							VarTempInt16:=8;
						END_IF
						IF(VarMastTempLoopCount>10)THEN    //取10次循环
							IF(VarMastA>-VarTempInt16) THEN
								VarMastA :=VarMastA - 1;
							ELSE
								VarMastA := -VarTempInt16;
							END_IF
							VarMastTempLoopCount:=0;
						END_IF
						VarMastTempLoopCount:=VarMastTempLoopCount + 1;
						VarMastB := VarMastA;
					ELSIF(VarAngleYDelta<-10)THEN
						IF(VarAngleYDelta<-30)THEN
							VarTempInt16:=16;
						ELSE
							VarTempInt16:=8;
						END_IF
						IF(VarMastTempLoopCount>10)THEN    //取10次循环
							IF(VarMastA<-VarTempInt16) THEN
								VarMastA :=VarMastA + 1;
							ELSE
								VarMastA := VarTempInt16;
							END_IF
							VarMastTempLoopCount:=0;
						END_IF
						VarMastTempLoopCount:=VarMastTempLoopCount + 1;
						VarMastB := VarMastA;
					ELSE
						VarMastA:= 0;
						VarMastB:= 0;
					END_IF
				END_CASE
			END_IF
		END_IF
	ELSE
		VarMastA := 0;
		VarMastB := 0;
	END_IF
	//自动调平OK时间
	IF(VarMastWorkMode=3 AND VarAngleXDelta>=-10 AND 
		VarAngleXDelta<=10 AND VarAngleYDelta>=-10 AND VarAngleYDelta<=10) THEN
		VarMastAutoOk_1:=TRUE;
	ELSE
		VarMastAutoOk_1:=FALSE;
	END_IF
			
	MastAutoTime(IN:=VarMastAutoOk_1,PT:=T#2S);
	VarMastAutoOk:=MastAutoTime.Q;
	
	//按下电手柄使能开关,自动退出自动模式
	IF(DIH_JOY) OR VarMastAutoOk THEN
		VarMastAutoEnable := FALSE;
		VarMastManuEnable := TRUE;
	END_IF
	
	//不能同时为零
	IF(NOT(VarMastManuEnable) AND NOT(VarMastAutoEnable))THEN
		VarMastManuEnable := TRUE;
		VarMastAutoEnable := FALSE;
	END_IF
	
	//作业模式只有手动
	IF(CANI_WorkModeSwitch)THEN
		VarMastManuEnable := TRUE;
		VarMastAutoEnable := FALSE;
	END_IF
	
	//自动模式,5.0度范围内
	IF( (VarAngleXDelta>=-500 AND VarAngleXDelta<=500) AND (VarAngleYDelta>=-500 AND VarAngleYDelta<=500))THEN
		VarAutoTiaoPingTiaoJian := TRUE;
	ELSE
		VarAutoTiaoPingTiaoJian := FALSE;
		IF(VarMastAutoEnable)THEN
			IF(VarAngleXDelta<-620 OR VarAngleXDelta>620 OR VarAngleYDelta<-620 OR VarAngleYDelta>620)THEN
				VarMastAutoEnable:= FALSE;
			END_IF
		ELSE
			VarMastAutoEnable := FALSE;	
		END_IF
	END_IF
	
	IF(CANI_Button_LEVER_Auto AND NOT(CANI_Button_LEVER_AutoLast))THEN
		VarMastAutoEnable := TRUE;
		VarMastManuEnable := FALSE;
	END_IF
	
	IF((NOT CANI_WorkModeSwitch) AND VarMastAutoEnable AND VarAutoTiaoPingTiaoJian)THEN
		VarMastWorkMode := 3; 
	END_IF
	
	//手动模式
	IF(CANI_Button_LEVER_Manual AND NOT(CANI_Button_LEVER_ManualLast)) THEN
		VarMastAutoEnable := FALSE;
		VarMastManuEnable := TRUE;
	END_IF
	IF(NOT CANI_WorkModeSwitch AND VarMastManuEnable) THEN
		VarMastWorkMode := 2;
	END_IF
	
	//限位模式
	IF(PAR_ControlValue<>9999) THEN
		IF((NOT DIH_SQ5) OR NOT(DIH_SQ6) OR TooHighY)THEN
			VarMastWorkMode := 1;
		END_IF
		VarMastLimitCancel := FALSE;
	ELSE
		IF(TooHighY)THEN
			VarMastWorkMode := 1;
			VarMastLimitCancel := FALSE;
		ELSE
			VarMastLimitCancel := TRUE;
		END_IF
	END_IF
	
	IF(NOT DIH_SQ5)THEN
		VarMastLimitState := 1;//左限位
	ELSIF(NOT DIH_SQ6)THEN
		VarMastLimitState := 2;//右限位
	ELSE
		VarMastLimitState := 0;
	END_IF
	
	IF(CANI_WorkModeSwitch AND VarMastWorkMode=3)THEN
			VarMastWorkMode := 2;
			VarMastManuEnable := TRUE;
			VarMastAutoEnable := FALSE;
	END_IF
	
	IF(DIH_JOY AND ((ABS(VarJoyX)>100) OR (ABS(VarJoyY)>100)) AND VarMastWorkMode=3)THEN
			VarMastWorkMode := 2;
			VarMastManuEnable := TRUE;
			VarMastAutoEnable := FALSE;
	END_IF
	
		//自动找垂步骤初值
	IF(VarMastWorkMode<>3)THEN
		VarMastAutoStep := 0;
		VarMastAutoEnable := FALSE;
	END_IF
	//更新标志
	CANI_Button_LEVER_AutoLast := CANI_Button_LEVER_Auto;
	CANI_Button_LEVER_ManualLast := CANI_Button_LEVER_Manual;

END_PROGRAM

// StandardPLC/Application/CAIJI/censor_cali
FUNCTION_BLOCK censor_cali
VAR_INPUT
	AI_ANGLE_X_c:UINT;
	AI_ANGLE_Y_c:UINT;
END_VAR
VAR_OUTPUT
	TooError_angle: BOOL;
END_VAR
VAR	
	ANGLE_X: INT;
	ANGLE_Y: INT;
	AngleX: ANGLE_CAIJI_X;
	AngleY: ANGLE_CAIJI_Y;
	TooLow_Water_Tem: BOOL;
	TooLow_hyd_Tem: BOOL;
	TooLow_lub_pressure: BOOL;
	TooHigh_hyd_tem: BOOL;
	TooHigh_water_tem: BOOL;
	FUEL_LEVER1: FUEL_LEVEL;
	TooLow_FUEL_LEVEL: BOOL;
	HYD_OIL_TEM1: HYD_OIL_TEM;
	CANO_TooError_ANGLE_X: BOOL;
	CANO_TooError_ANGLE_Y: BOOL;
	TooHighY_TEST: BOOL;
	P11_mainpump1:PRESSURE;
	P12_mainpump2:PRESSURE;
	P1_JiaYa:PRESSURE;
	P2_donglitou:PRESSURE;
	P3_mainwinch:PRESSURE;
	P6_fubeng:PRESSURE;
	P7_Pilot_PRESSURE:PRESSURE;
	P8_Rotation_PRESSURE: PRESSURE;
	MainTension:Tension;
	SaveEngine_PAcPre: PRESSURE;
	SaveEngine_PAtomsPre: PRESSURE;
	SaveEngine_PM1Pre: PRESSURE;
	SaveEngine_PM2Pre: PRESSURE;
(*	Flow_Q1: Flow;
	Flow_Q2: Flow;
	Flow_QAc: Flow;
	Flow_QM1: Flow;*)
END_VAR

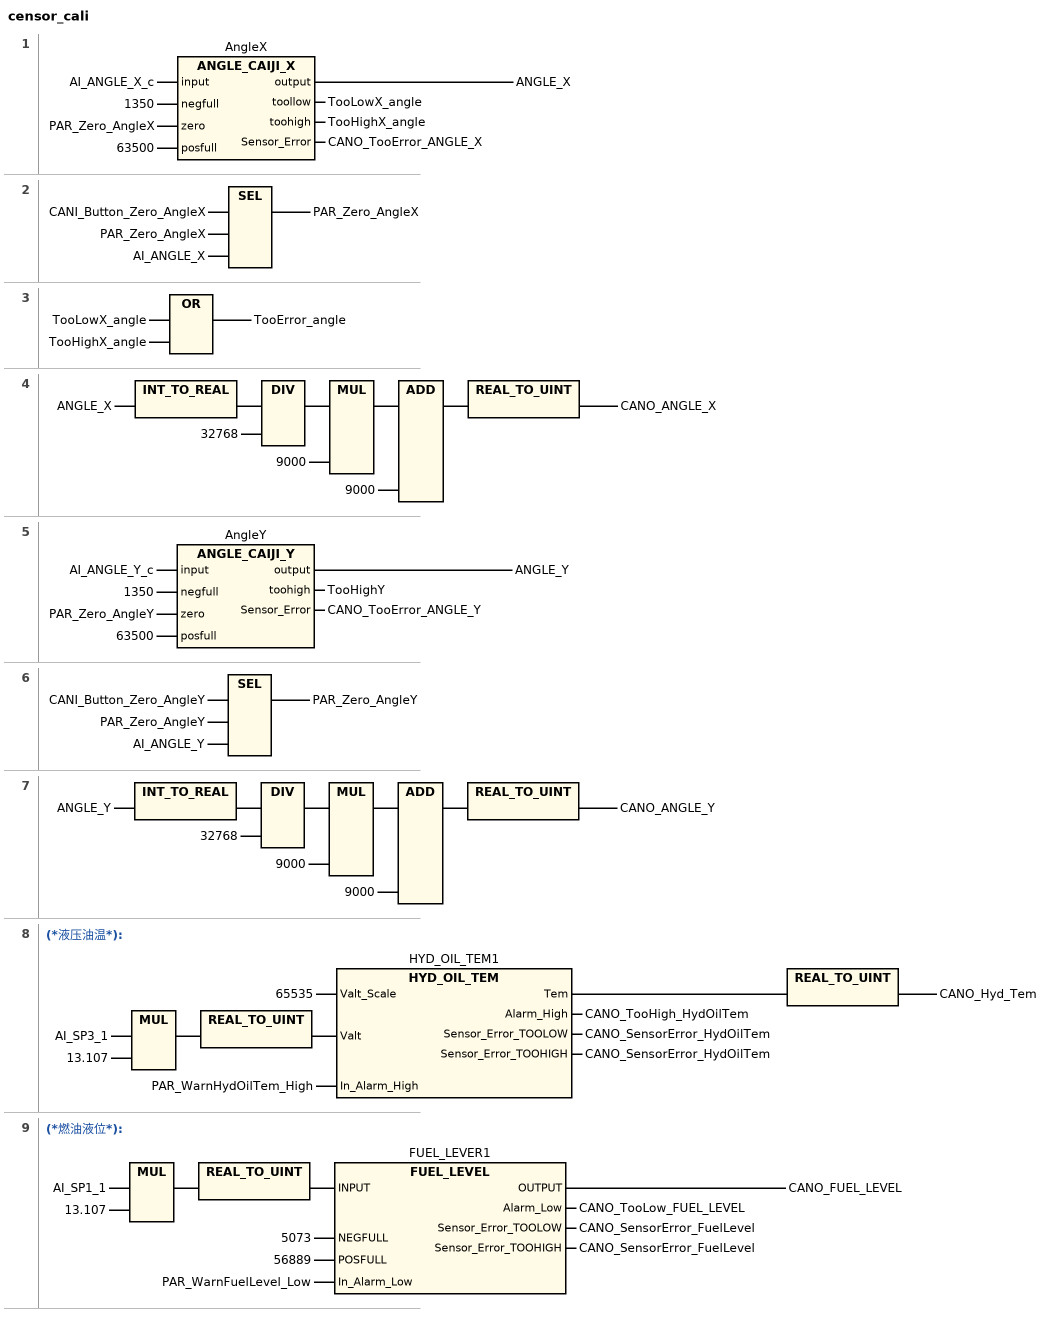
// NETWORK 1
AngleX(
    input := AI_ANGLE_X_c,
    negfull := 1350,
    zero := PAR_Zero_AngleX,
    posfull := 63500,
    toollow => TooLowX_angle,
    toohigh => TooHighX_angle,
    Sensor_Error => CANO_TooError_ANGLE_X); // ANGLE_CAIJI_X
ANGLE_X := AngleX.output;

// NETWORK 2
PAR_Zero_AngleX := SEL(CANI_Button_Zero_AngleX, PAR_Zero_AngleX, AI_ANGLE_X);

// NETWORK 3
TooError_angle := TooLowX_angle OR TooHighX_angle;

// NETWORK 4
CANO_ANGLE_X := REAL_TO_UINT((INT_TO_REAL(ANGLE_X) / 32768) * 9000 + 9000);

// NETWORK 5
AngleY(
    input := AI_ANGLE_Y_c,
    negfull := 1350,
    zero := PAR_Zero_AngleY,
    posfull := 63500,
    toohigh => TooHighY,
    Sensor_Error => CANO_TooError_ANGLE_Y); // ANGLE_CAIJI_Y
ANGLE_Y := AngleY.output;

// NETWORK 6
PAR_Zero_AngleY := SEL(CANI_Button_Zero_AngleY, PAR_Zero_AngleY, AI_ANGLE_Y);

// NETWORK 7
CANO_ANGLE_Y := REAL_TO_UINT((INT_TO_REAL(ANGLE_Y) / 32768) * 9000 + 9000);

// NETWORK 8
// label: (*液压油温*)
HYD_OIL_TEM1(
    Valt_Scale := 65535,
    Valt := REAL_TO_UINT(AI_SP3_1 * 13.107),
    In_Alarm_High := PAR_WarnHydOilTem_High,
    Alarm_High => CANO_TooHigh_HydOilTem,
    Sensor_Error_TOOLOW => CANO_SensorError_HydOilTem,
    Sensor_Error_TOOHIGH => CANO_SensorError_HydOilTem); // HYD_OIL_TEM
CANO_Hyd_Tem := REAL_TO_UINT(HYD_OIL_TEM1.Tem);

// NETWORK 9
// label: (*燃油液位*)
FUEL_LEVER1(
    INPUT := REAL_TO_UINT(AI_SP1_1 * 13.107),
    NEGFULL := 5073,
    POSFULL := 56889,
    In_Alarm_Low := PAR_WarnFuelLevel_Low,
    Alarm_Low => CANO_TooLow_FUEL_LEVEL,
    Sensor_Error_TOOLOW => CANO_SensorError_FuelLevel,
    Sensor_Error_TOOHIGH => CANO_SensorError_FuelLevel); // FUEL_LEVEL
CANO_FUEL_LEVEL := FUEL_LEVER1.OUTPUT;

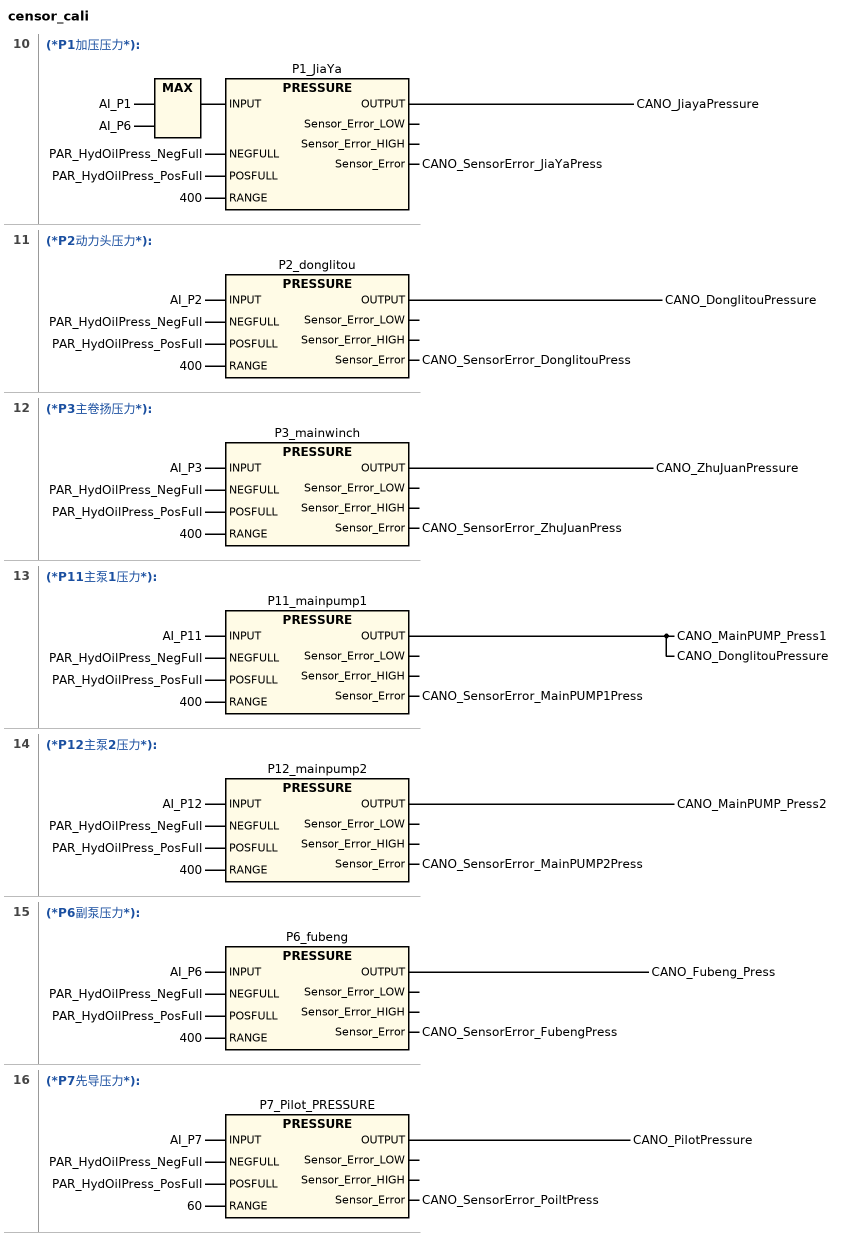
// NETWORK 10
// label: (*P1加压压力*)
P1_JiaYa(
    INPUT := MAX(AI_P1, AI_P6),
    NEGFULL := PAR_HydOilPress_NegFull,
    POSFULL := PAR_HydOilPress_PosFull,
    RANGE := 400,
    Sensor_Error => CANO_SensorError_JiaYaPress); // PRESSURE
CANO_JiayaPressure := P1_JiaYa.OUTPUT;

// NETWORK 11
// label: (*P2动力头压力*)
P2_donglitou(
    INPUT := AI_P2,
    NEGFULL := PAR_HydOilPress_NegFull,
    POSFULL := PAR_HydOilPress_PosFull,
    RANGE := 400,
    Sensor_Error => CANO_SensorError_DonglitouPress); // PRESSURE
CANO_DonglitouPressure := P2_donglitou.OUTPUT;

// NETWORK 12
// label: (*P3主卷扬压力*)
P3_mainwinch(
    INPUT := AI_P3,
    NEGFULL := PAR_HydOilPress_NegFull,
    POSFULL := PAR_HydOilPress_PosFull,
    RANGE := 400,
    Sensor_Error => CANO_SensorError_ZhuJuanPress); // PRESSURE
CANO_ZhuJuanPressure := P3_mainwinch.OUTPUT;

// NETWORK 13
// label: (*P11主泵1压力*)
P11_mainpump1(
    INPUT := AI_P11,
    NEGFULL := PAR_HydOilPress_NegFull,
    POSFULL := PAR_HydOilPress_PosFull,
    RANGE := 400,
    Sensor_Error => CANO_SensorError_MainPUMP1Press); // PRESSURE
CANO_MainPUMP_Press1 := P11_mainpump1.OUTPUT;
CANO_DonglitouPressure := P11_mainpump1.OUTPUT;

// NETWORK 14
// label: (*P12主泵2压力*)
P12_mainpump2(
    INPUT := AI_P12,
    NEGFULL := PAR_HydOilPress_NegFull,
    POSFULL := PAR_HydOilPress_PosFull,
    RANGE := 400,
    Sensor_Error => CANO_SensorError_MainPUMP2Press); // PRESSURE
CANO_MainPUMP_Press2 := P12_mainpump2.OUTPUT;

// NETWORK 15
// label: (*P6副泵压力*)
P6_fubeng(
    INPUT := AI_P6,
    NEGFULL := PAR_HydOilPress_NegFull,
    POSFULL := PAR_HydOilPress_PosFull,
    RANGE := 400,
    Sensor_Error => CANO_SensorError_FubengPress); // PRESSURE
CANO_Fubeng_Press := P6_fubeng.OUTPUT;

// NETWORK 16
// label: (*P7先导压力*)
P7_Pilot_PRESSURE(
    INPUT := AI_P7,
    NEGFULL := PAR_HydOilPress_NegFull,
    POSFULL := PAR_HydOilPress_PosFull,
    RANGE := 60,
    Sensor_Error => CANO_SensorError_PoiltPress); // PRESSURE
CANO_PilotPressure := P7_Pilot_PRESSURE.OUTPUT;

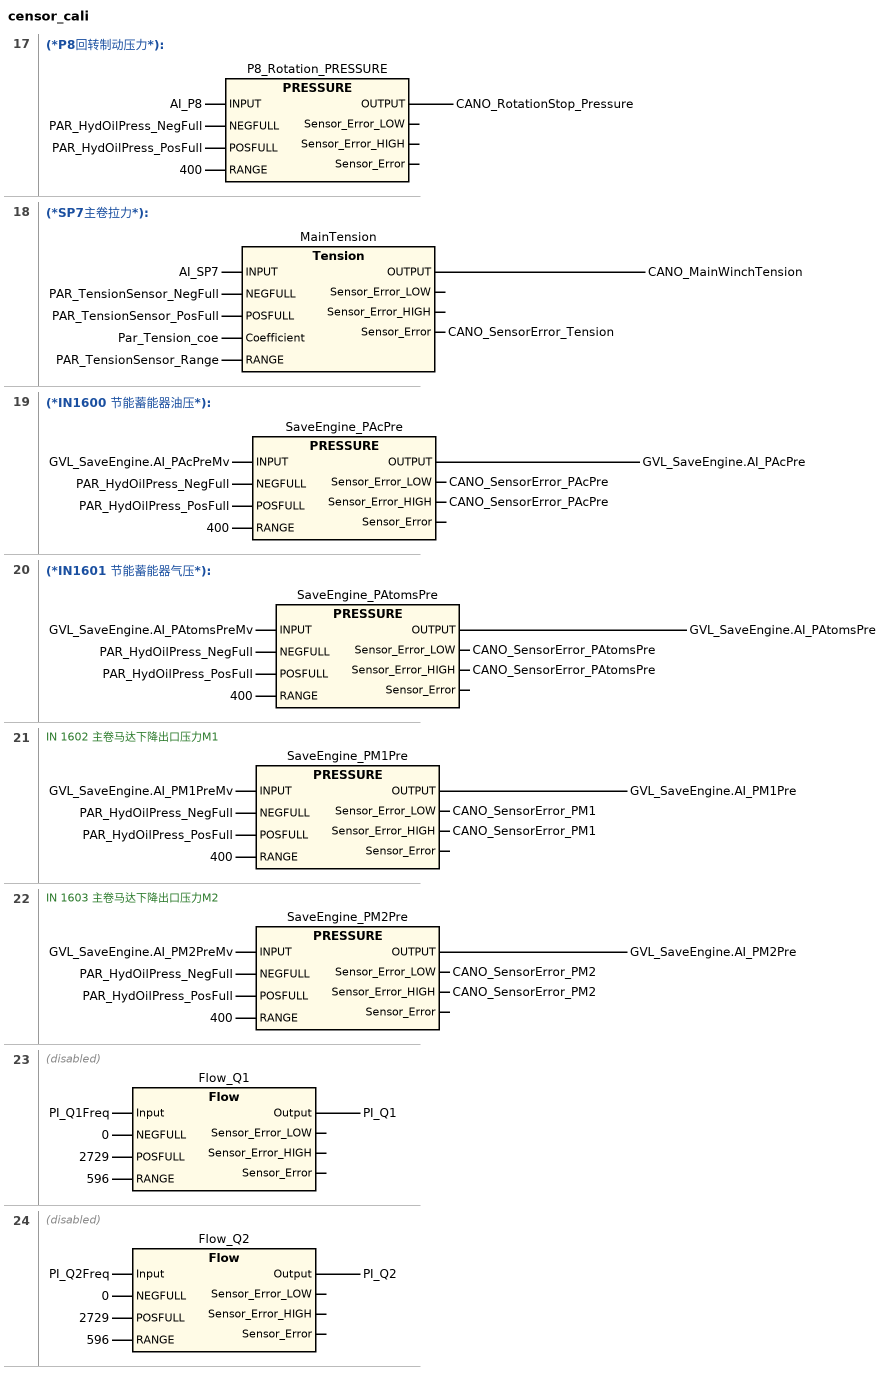
// NETWORK 17
// label: (*P8回转制动压力*)
P8_Rotation_PRESSURE(
    INPUT := AI_P8,
    NEGFULL := PAR_HydOilPress_NegFull,
    POSFULL := PAR_HydOilPress_PosFull,
    RANGE := 400); // PRESSURE
CANO_RotationStop_Pressure := P8_Rotation_PRESSURE.OUTPUT;

// NETWORK 18
// label: (*SP7主卷拉力*)
MainTension(
    INPUT := AI_SP7,
    NEGFULL := PAR_TensionSensor_NegFull,
    POSFULL := PAR_TensionSensor_PosFull,
    Coefficient := Par_Tension_coe,
    RANGE := PAR_TensionSensor_Range,
    Sensor_Error => CANO_SensorError_Tension); // Tension
CANO_MainWinchTension := MainTension.OUTPUT;

// NETWORK 19
// label: (*IN1600 节能蓄能器油压*)
SaveEngine_PAcPre(
    INPUT := GVL_SaveEngine.AI_PAcPreMv,
    NEGFULL := PAR_HydOilPress_NegFull,
    POSFULL := PAR_HydOilPress_PosFull,
    RANGE := 400,
    Sensor_Error_LOW => CANO_SensorError_PAcPre,
    Sensor_Error_HIGH => CANO_SensorError_PAcPre); // PRESSURE
GVL_SaveEngine.AI_PAcPre := SaveEngine_PAcPre.OUTPUT;

